ABB RAPID module: WeldProgram.mod

MODULE WeldProgram

    ! =========================
    ! ======= SAFE POS ========
    ! =========================
    PERS robtarget pSafeS1 := [[82.84,919.33,1175.90],[0.326608,0.635474,-0.637382,0.288521],[0,0,-1,0],[9E9,9E9,9E9,9E9,9E9,9E9]];
    PERS robtarget pSafeS1Weld := [[82.84,919.33,1175.90],[0.326608,0.635474,-0.637382,0.288521],[0,0,-1,0],[9E9,9E9,9E9,9E9,9E9,9E9]];
    PERS robtarget pSetup  := [[82.84,919.33,1175.90],[0.326608,0.635474,-0.637382,0.288521],[0,0,-1,0],[9E9,9E9,9E9,9E9,9E9,9E9]];
    PERS robtarget pBullseye := [[82.84,919.33,1175.90],[0.326608,0.635474,-0.637382,0.288521],[0,0,-1,0],[9E9,9E9,9E9,9E9,9E9,9E9]];
    PERS robtarget pFixtureCheck := [[82.84,919.33,1175.90],[0.326608,0.635474,-0.637382,0.288521],[0,0,-1,0],[9E9,9E9,9E9,9E9,9E9,9E9]];

    ! =========================
    ! == DEFAULT WELD DATA ====
    ! =========================
    PERS seamdata cSeamDefault := [1,1,[1,0,14,127,0,0,0,0,0],0,0,0,0,0,[0,0,0,0,0,0,0,0,0],0,0,[0,0,0,0,0,0,0,0,0],0,0,[0,0,0,0,0,0,0,0,0],0];
    PERS welddata cWeldDefault := [6.90033,6.90033,[1,0,19,110.71,0,0,0,0,0],[0,0,18.5,110.71,0,0,0,0,0]];
    PERS weavedata cWeaveDefault := [1,1,3.81,5.08,1.778,0,0,0,0,0,0,0,0,0,0];

    ! =========================
    ! === PART METADATA =======
    ! =========================
    PERS string partNameP01 := "Part 1";
    PERS string partNameP02 := "Part 2";
    PERS string partNameP03 := "Part 3";
    PERS string partNameP04 := "Part 4";
    PERS string partNameP05 := "Part 5";
    PERS string partNameP06 := "Part 6";
    PERS bool partEnabledP01 := TRUE;
    PERS bool partEnabledP02 := TRUE;
    PERS bool partEnabledP03 := TRUE;
    PERS bool partEnabledP04 := TRUE;
    PERS bool partEnabledP05 := TRUE;
    PERS bool partEnabledP06 := TRUE;

    ! =========================
    ! ====== SPEEDS ===========
    ! =========================
    PERS speeddata vPreviewArcStart := [5,500,5000,1000];
    PERS speeddata vPreviewArcEnd := [5,500,5000,1000];
    PERS speeddata vPreviewApproach := [5,500,5000,1000];
    PERS speeddata vPreviewRetract := [5,500,5000,1000];
    PERS speeddata vPreviewTrans := [5,500,5000,1000];
    PERS speeddata vProdArcStart := [100,500,5000,1000];
    PERS speeddata vProdArcEnd := [100,500,5000,1000];
    PERS speeddata vProdApproach := [100,500,5000,1000];
    PERS speeddata vProdRetract := [100,500,5000,1000];
    PERS speeddata vProdTrans := [100,500,5000,1000];

    ! =========================
    ! == ORIENTATION POSES ====
    ! =========================
    PERS robtarget pOri_Left := [[-322.341,524.952,62.8015],[0.119487,0.856675,-0.263973,0.426789],[1,-1,-1,0],[9E+09,9E+09,9E+09,9E+09,9E+09,9E+09]];
    PERS robtarget pOri_Right:= [[-338.053,523.699,62.2846],[0.437822,0.2846,-0.843699,0.124444],[1,0,0,0],[9E+09,9E+09,9E+09,9E+09,9E+09,9E+09]];
    PERS robtarget pOri_Up   := [[-324.994,521.603,62.1105],[0.180394,0.831672,-0.360019,0.382317],[1,0,-1,0],[9E+09,9E+09,9E+09,9E+09,9E+09,9E+09]];
    PERS robtarget pOri_Down := [[-327.638,525.763,56.7062],[0.26234,-0.322639,0.903337,0.105184],[1,-1,2,0],[9E+09,9E+09,9E+09,9E+09,9E+09,9E+09]];
    PERS robtarget pOri_yMid := [[0,0,0],[1,0,0,0],[0,0,0,0],[9E9,9E9,9E9,9E9,9E9,9E9]];
    PERS robtarget pOri_xMid := [[0,0,0],[1,0,0,0],[0,0,0,0],[9E9,9E9,9E9,9E9,9E9,9E9]];

    ! =========================
    ! ===== PART FRAMES =======
    ! =========================
    PERS robtarget P01Origin := [[0,0,0],[1,0,0,0],[0,0,0,0],[9E9,9E9,9E9,9E9,9E9,9E9]];
    PERS robtarget P01Max    := [[0,0,0],[1,0,0,0],[0,0,0,0],[9E9,9E9,9E9,9E9,9E9,9E9]];
    PERS robtarget P01Zoff   := [[0,0,0],[1,0,0,0],[0,0,0,0],[9E9,9E9,9E9,9E9,9E9,9E9]];
    PERS wobjdata wobjP01 := [FALSE,TRUE,"",[[0,0,0],[1,0,0,0]],[[0,0,0],[1,0,0,0]]];
    PERS num nWeldsP01 := 5;

    PERS robtarget P02Origin := [[-1364.6,652.519,70.0999],[0.0320518,0.697908,-0.715468,-0.00179197],[1,-1,1,0],[9E+09,9E+09,9E+09,9E+09,9E+09,9E+09]];
    PERS robtarget P02Max    := [[-382.936,1483.05,51.6185],[0.0320653,0.697883,-0.715492,-0.00180713],[1,-2,1,0],[9E+09,9E+09,9E+09,9E+09,9E+09,9E+09]];
    PERS robtarget P02Zoff   := [[-392.282,1373.57,51.6146],[0.032034,0.697931,-0.715446,-0.00178465],[1,-2,1,0],[9E+09,9E+09,9E+09,9E+09,9E+09,9E+09]];
    PERS wobjdata wobjP02 := [FALSE,TRUE,"",[[-1364.6,652.519,70.0999],[0.0320518,0.697908,-0.715468,-0.00179197]],[[-392.282,1373.57,51.6146],[0.032034,0.697931,-0.715446,-0.00178465]]];
    PERS num nWeldsP02 := 2;

    PERS robtarget P03Origin := [[0,0,0],[1,0,0,0],[0,0,0,0],[9E9,9E9,9E9,9E9,9E9,9E9]];
    PERS robtarget P03Max    := [[0,0,0],[1,0,0,0],[0,0,0,0],[9E9,9E9,9E9,9E9,9E9,9E9]];
    PERS robtarget P03Zoff   := [[0,0,0],[1,0,0,0],[0,0,0,0],[9E9,9E9,9E9,9E9,9E9,9E9]];
    PERS wobjdata wobjP03 := [FALSE,TRUE,"",[[0,0,0],[1,0,0,0]],[[0,0,0],[1,0,0,0]]];
    PERS num nWeldsP03 := 0;

    PERS robtarget P04Origin := [[0,0,0],[1,0,0,0],[0,0,0,0],[9E9,9E9,9E9,9E9,9E9,9E9]];
    PERS robtarget P04Max    := [[0,0,0],[1,0,0,0],[0,0,0,0],[9E9,9E9,9E9,9E9,9E9,9E9]];
    PERS robtarget P04Zoff   := [[0,0,0],[1,0,0,0],[0,0,0,0],[9E9,9E9,9E9,9E9,9E9,9E9]];
    PERS wobjdata wobjP04 := [FALSE,TRUE,"",[[0,0,0],[1,0,0,0]],[[0,0,0],[1,0,0,0]]];
    PERS num nWeldsP04 := 0;

    PERS robtarget P05Origin := [[0,0,0],[1,0,0,0],[0,0,0,0],[9E9,9E9,9E9,9E9,9E9,9E9]];
    PERS robtarget P05Max    := [[0,0,0],[1,0,0,0],[0,0,0,0],[9E9,9E9,9E9,9E9,9E9,9E9]];
    PERS robtarget P05Zoff   := [[0,0,0],[1,0,0,0],[0,0,0,0],[9E9,9E9,9E9,9E9,9E9,9E9]];
    PERS wobjdata wobjP05 := [FALSE,TRUE,"",[[0,0,0],[1,0,0,0]],[[0,0,0],[1,0,0,0]]];
    PERS num nWeldsP05 := 0;

    PERS robtarget P06Origin := [[0,0,0],[1,0,0,0],[0,0,0,0],[9E9,9E9,9E9,9E9,9E9,9E9]];
    PERS robtarget P06Max    := [[0,0,0],[1,0,0,0],[0,0,0,0],[9E9,9E9,9E9,9E9,9E9,9E9]];
    PERS robtarget P06Zoff   := [[0,0,0],[1,0,0,0],[0,0,0,0],[9E9,9E9,9E9,9E9,9E9,9E9]];
    PERS wobjdata wobjP06 := [FALSE,TRUE,"",[[0,0,0],[1,0,0,0]],[[0,0,0],[1,0,0,0]]];
    PERS num nWeldsP06 := 0;

    ! =========================
    ! == WELD SLOT STORAGE ====
    ! =========================
    ! ---- P01 weld slots ----
    PERS bool P01W01_Used := TRUE;
    PERS num  P01W01_SubType := 22;
    PERS num  P01W01_ToolSel := 4;
    PERS num  P01W01_LenMM := 31.75;
    PERS robtarget P01W01_ArcStart := [[-1.72108,1549.32,-10.8357],[0.26234,-0.322639,0.903337,0.105184],[1,-1,2,0],[9E+09,9E+09,9E+09,9E+09,9E+09,9E+09]];
    PERS robtarget P01W01_ArcEnd   := [[30.0289,1549.32,-10.8357],[0.26234,-0.322639,0.903337,0.105184],[1,-1,2,0],[9E+09,9E+09,9E+09,9E+09,9E+09,9E+09]];
    PERS robtarget P01W01_Approach := [[-4.26108,1546.78,-8.29572],[0.26234,-0.322639,0.903337,0.105184],[1,-1,2,0],[9E+09,9E+09,9E+09,9E+09,9E+09,9E+09]];
    PERS robtarget P01W01_Retract  := [[27.4889,1546.78,-8.29572],[0.26234,-0.322639,0.903337,0.105184],[1,-1,2,0],[9E+09,9E+09,9E+09,9E+09,9E+09,9E+09]];
    PERS robtarget P01W01_Trans    := [[27.4889,1546.78,245.704],[0.26234,-0.322639,0.903337,0.105184],[1,-1,2,0],[9E+09,9E+09,9E+09,9E+09,9E+09,9E+09]];
    PERS bool P01W02_Used := TRUE;
    PERS num  P01W02_SubType := 21;
    PERS num  P01W02_ToolSel := 3;
    PERS num  P01W02_LenMM := 31.75;
    PERS robtarget P01W02_ArcStart := [[-313.218,545.116,2.61322],[0.180394,0.831672,-0.360019,0.382317],[1,0,-1,0],[9E+09,9E+09,9E+09,9E+09,9E+09,9E+09]];
    PERS robtarget P01W02_ArcEnd   := [[-281.468,545.116,2.61322],[0.180394,0.831672,-0.360019,0.382317],[1,0,-1,0],[9E+09,9E+09,9E+09,9E+09,9E+09,9E+09]];
    PERS robtarget P01W02_Approach := [[-315.758,547.656,5.15322],[0.180394,0.831672,-0.360019,0.382317],[1,0,-1,0],[9E+09,9E+09,9E+09,9E+09,9E+09,9E+09]];
    PERS robtarget P01W02_Retract  := [[-284.008,547.656,5.15322],[0.180394,0.831672,-0.360019,0.382317],[1,0,-1,0],[9E+09,9E+09,9E+09,9E+09,9E+09,9E+09]];
    PERS robtarget P01W02_Trans    := [[-284.008,547.656,259.153],[0.180394,0.831672,-0.360019,0.382317],[1,0,-1,0],[9E+09,9E+09,9E+09,9E+09,9E+09,9E+09]];
    PERS bool P01W03_Used := TRUE;
    PERS num  P01W03_SubType := 21;
    PERS num  P01W03_ToolSel := 3;
    PERS num  P01W03_LenMM := 31.75;
    PERS robtarget P01W03_ArcStart := [[4.28168,545.116,2.61322],[0.180394,0.831672,-0.360019,0.382317],[1,0,-1,0],[9E+09,9E+09,9E+09,9E+09,9E+09,9E+09]];
    PERS robtarget P01W03_ArcEnd   := [[36.0317,545.116,2.61322],[0.180394,0.831672,-0.360019,0.382317],[1,0,-1,0],[9E+09,9E+09,9E+09,9E+09,9E+09,9E+09]];
    PERS robtarget P01W03_Approach := [[1.74168,547.656,5.15322],[0.180394,0.831672,-0.360019,0.382317],[1,0,-1,0],[9E+09,9E+09,9E+09,9E+09,9E+09,9E+09]];
    PERS robtarget P01W03_Retract  := [[33.4917,547.656,5.15322],[0.180394,0.831672,-0.360019,0.382317],[1,0,-1,0],[9E+09,9E+09,9E+09,9E+09,9E+09,9E+09]];
    PERS robtarget P01W03_Trans    := [[33.4917,547.656,259.153],[0.180394,0.831672,-0.360019,0.382317],[1,0,-1,0],[9E+09,9E+09,9E+09,9E+09,9E+09,9E+09]];
    PERS bool P01W04_Used := TRUE;
    PERS num  P01W04_SubType := 21;
    PERS num  P01W04_ToolSel := 3;
    PERS num  P01W04_LenMM := 31.75;
    PERS robtarget P01W04_ArcStart := [[861.532,545.116,2.61322],[0.180394,0.831672,-0.360019,0.382317],[1,0,-1,0],[9E+09,9E+09,9E+09,9E+09,9E+09,9E+09]];
    PERS robtarget P01W04_ArcEnd   := [[893.282,545.116,2.61322],[0.180394,0.831672,-0.360019,0.382317],[1,0,-1,0],[9E+09,9E+09,9E+09,9E+09,9E+09,9E+09]];
    PERS robtarget P01W04_Approach := [[858.992,547.656,5.15322],[0.180394,0.831672,-0.360019,0.382317],[1,0,-1,0],[9E+09,9E+09,9E+09,9E+09,9E+09,9E+09]];
    PERS robtarget P01W04_Retract  := [[890.742,547.656,5.15322],[0.180394,0.831672,-0.360019,0.382317],[1,0,-1,0],[9E+09,9E+09,9E+09,9E+09,9E+09,9E+09]];
    PERS robtarget P01W04_Trans    := [[890.742,547.656,259.153],[0.180394,0.831672,-0.360019,0.382317],[1,0,-1,0],[9E+09,9E+09,9E+09,9E+09,9E+09,9E+09]];
    PERS bool P01W05_Used := TRUE;
    PERS num  P01W05_SubType := 21;
    PERS num  P01W05_ToolSel := 3;
    PERS num  P01W05_LenMM := 31.75;
    PERS robtarget P01W05_ArcStart := [[1166.33,545.116,2.61322],[0.180394,0.831672,-0.360019,0.382317],[1,0,-1,0],[9E+09,9E+09,9E+09,9E+09,9E+09,9E+09]];
    PERS robtarget P01W05_ArcEnd   := [[1198.08,545.116,2.61322],[0.180394,0.831672,-0.360019,0.382317],[1,0,-1,0],[9E+09,9E+09,9E+09,9E+09,9E+09,9E+09]];
    PERS robtarget P01W05_Approach := [[1163.79,547.656,5.15322],[0.180394,0.831672,-0.360019,0.382317],[1,0,-1,0],[9E+09,9E+09,9E+09,9E+09,9E+09,9E+09]];
    PERS robtarget P01W05_Retract  := [[1195.54,547.656,5.15322],[0.180394,0.831672,-0.360019,0.382317],[1,0,-1,0],[9E+09,9E+09,9E+09,9E+09,9E+09,9E+09]];
    PERS robtarget P01W05_Trans    := [[1195.54,547.656,259.153],[0.180394,0.831672,-0.360019,0.382317],[1,0,-1,0],[9E+09,9E+09,9E+09,9E+09,9E+09,9E+09]];
    PERS bool P01W06_Used := FALSE;
    PERS num  P01W06_SubType := 0;
    PERS num  P01W06_ToolSel := 0;
    PERS num  P01W06_LenMM := 0;
    PERS robtarget P01W06_ArcStart := [[0,0,0],[1,0,0,0],[0,0,0,0],[9E9,9E9,9E9,9E9,9E9,9E9]];
    PERS robtarget P01W06_ArcEnd   := [[0,0,0],[1,0,0,0],[0,0,0,0],[9E9,9E9,9E9,9E9,9E9,9E9]];
    PERS robtarget P01W06_Approach := [[0,0,0],[1,0,0,0],[0,0,0,0],[9E9,9E9,9E9,9E9,9E9,9E9]];
    PERS robtarget P01W06_Retract  := [[0,0,0],[1,0,0,0],[0,0,0,0],[9E9,9E9,9E9,9E9,9E9,9E9]];
    PERS robtarget P01W06_Trans    := [[0,0,0],[1,0,0,0],[0,0,0,0],[9E9,9E9,9E9,9E9,9E9,9E9]];
    PERS bool P01W07_Used := FALSE;
    PERS num  P01W07_SubType := 0;
    PERS num  P01W07_ToolSel := 0;
    PERS num  P01W07_LenMM := 0;
    PERS robtarget P01W07_ArcStart := [[0,0,0],[1,0,0,0],[0,0,0,0],[9E9,9E9,9E9,9E9,9E9,9E9]];
    PERS robtarget P01W07_ArcEnd   := [[0,0,0],[1,0,0,0],[0,0,0,0],[9E9,9E9,9E9,9E9,9E9,9E9]];
    PERS robtarget P01W07_Approach := [[0,0,0],[1,0,0,0],[0,0,0,0],[9E9,9E9,9E9,9E9,9E9,9E9]];
    PERS robtarget P01W07_Retract  := [[0,0,0],[1,0,0,0],[0,0,0,0],[9E9,9E9,9E9,9E9,9E9,9E9]];
    PERS robtarget P01W07_Trans    := [[0,0,0],[1,0,0,0],[0,0,0,0],[9E9,9E9,9E9,9E9,9E9,9E9]];
    PERS bool P01W08_Used := FALSE;
    PERS num  P01W08_SubType := 0;
    PERS num  P01W08_ToolSel := 0;
    PERS num  P01W08_LenMM := 0;
    PERS robtarget P01W08_ArcStart := [[0,0,0],[1,0,0,0],[0,0,0,0],[9E9,9E9,9E9,9E9,9E9,9E9]];
    PERS robtarget P01W08_ArcEnd   := [[0,0,0],[1,0,0,0],[0,0,0,0],[9E9,9E9,9E9,9E9,9E9,9E9]];
    PERS robtarget P01W08_Approach := [[0,0,0],[1,0,0,0],[0,0,0,0],[9E9,9E9,9E9,9E9,9E9,9E9]];
    PERS robtarget P01W08_Retract  := [[0,0,0],[1,0,0,0],[0,0,0,0],[9E9,9E9,9E9,9E9,9E9,9E9]];
    PERS robtarget P01W08_Trans    := [[0,0,0],[1,0,0,0],[0,0,0,0],[9E9,9E9,9E9,9E9,9E9,9E9]];
    PERS bool P01W09_Used := FALSE;
    PERS num  P01W09_SubType := 0;
    PERS num  P01W09_ToolSel := 0;
    PERS num  P01W09_LenMM := 0;
    PERS robtarget P01W09_ArcStart := [[0,0,0],[1,0,0,0],[0,0,0,0],[9E9,9E9,9E9,9E9,9E9,9E9]];
    PERS robtarget P01W09_ArcEnd   := [[0,0,0],[1,0,0,0],[0,0,0,0],[9E9,9E9,9E9,9E9,9E9,9E9]];
    PERS robtarget P01W09_Approach := [[0,0,0],[1,0,0,0],[0,0,0,0],[9E9,9E9,9E9,9E9,9E9,9E9]];
    PERS robtarget P01W09_Retract  := [[0,0,0],[1,0,0,0],[0,0,0,0],[9E9,9E9,9E9,9E9,9E9,9E9]];
    PERS robtarget P01W09_Trans    := [[0,0,0],[1,0,0,0],[0,0,0,0],[9E9,9E9,9E9,9E9,9E9,9E9]];
    PERS bool P01W10_Used := FALSE;
    PERS num  P01W10_SubType := 0;
    PERS num  P01W10_ToolSel := 0;
    PERS num  P01W10_LenMM := 0;
    PERS robtarget P01W10_ArcStart := [[0,0,0],[1,0,0,0],[0,0,0,0],[9E9,9E9,9E9,9E9,9E9,9E9]];
    PERS robtarget P01W10_ArcEnd   := [[0,0,0],[1,0,0,0],[0,0,0,0],[9E9,9E9,9E9,9E9,9E9,9E9]];
    PERS robtarget P01W10_Approach := [[0,0,0],[1,0,0,0],[0,0,0,0],[9E9,9E9,9E9,9E9,9E9,9E9]];
    PERS robtarget P01W10_Retract  := [[0,0,0],[1,0,0,0],[0,0,0,0],[9E9,9E9,9E9,9E9,9E9,9E9]];
    PERS robtarget P01W10_Trans    := [[0,0,0],[1,0,0,0],[0,0,0,0],[9E9,9E9,9E9,9E9,9E9,9E9]];
    PERS bool P01W11_Used := FALSE;
    PERS num  P01W11_SubType := 0;
    PERS num  P01W11_ToolSel := 0;
    PERS num  P01W11_LenMM := 0;
    PERS robtarget P01W11_ArcStart := [[0,0,0],[1,0,0,0],[0,0,0,0],[9E9,9E9,9E9,9E9,9E9,9E9]];
    PERS robtarget P01W11_ArcEnd   := [[0,0,0],[1,0,0,0],[0,0,0,0],[9E9,9E9,9E9,9E9,9E9,9E9]];
    PERS robtarget P01W11_Approach := [[0,0,0],[1,0,0,0],[0,0,0,0],[9E9,9E9,9E9,9E9,9E9,9E9]];
    PERS robtarget P01W11_Retract  := [[0,0,0],[1,0,0,0],[0,0,0,0],[9E9,9E9,9E9,9E9,9E9,9E9]];
    PERS robtarget P01W11_Trans    := [[0,0,0],[1,0,0,0],[0,0,0,0],[9E9,9E9,9E9,9E9,9E9,9E9]];
    PERS bool P01W12_Used := FALSE;
    PERS num  P01W12_SubType := 0;
    PERS num  P01W12_ToolSel := 0;
    PERS num  P01W12_LenMM := 0;
    PERS robtarget P01W12_ArcStart := [[0,0,0],[1,0,0,0],[0,0,0,0],[9E9,9E9,9E9,9E9,9E9,9E9]];
    PERS robtarget P01W12_ArcEnd   := [[0,0,0],[1,0,0,0],[0,0,0,0],[9E9,9E9,9E9,9E9,9E9,9E9]];
    PERS robtarget P01W12_Approach := [[0,0,0],[1,0,0,0],[0,0,0,0],[9E9,9E9,9E9,9E9,9E9,9E9]];
    PERS robtarget P01W12_Retract  := [[0,0,0],[1,0,0,0],[0,0,0,0],[9E9,9E9,9E9,9E9,9E9,9E9]];
    PERS robtarget P01W12_Trans    := [[0,0,0],[1,0,0,0],[0,0,0,0],[9E9,9E9,9E9,9E9,9E9,9E9]];
    PERS bool P01W13_Used := FALSE;
    PERS num  P01W13_SubType := 0;
    PERS num  P01W13_ToolSel := 0;
    PERS num  P01W13_LenMM := 0;
    PERS robtarget P01W13_ArcStart := [[0,0,0],[1,0,0,0],[0,0,0,0],[9E9,9E9,9E9,9E9,9E9,9E9]];
    PERS robtarget P01W13_ArcEnd   := [[0,0,0],[1,0,0,0],[0,0,0,0],[9E9,9E9,9E9,9E9,9E9,9E9]];
    PERS robtarget P01W13_Approach := [[0,0,0],[1,0,0,0],[0,0,0,0],[9E9,9E9,9E9,9E9,9E9,9E9]];
    PERS robtarget P01W13_Retract  := [[0,0,0],[1,0,0,0],[0,0,0,0],[9E9,9E9,9E9,9E9,9E9,9E9]];
    PERS robtarget P01W13_Trans    := [[0,0,0],[1,0,0,0],[0,0,0,0],[9E9,9E9,9E9,9E9,9E9,9E9]];
    PERS bool P01W14_Used := FALSE;
    PERS num  P01W14_SubType := 0;
    PERS num  P01W14_ToolSel := 0;
    PERS num  P01W14_LenMM := 0;
    PERS robtarget P01W14_ArcStart := [[0,0,0],[1,0,0,0],[0,0,0,0],[9E9,9E9,9E9,9E9,9E9,9E9]];
    PERS robtarget P01W14_ArcEnd   := [[0,0,0],[1,0,0,0],[0,0,0,0],[9E9,9E9,9E9,9E9,9E9,9E9]];
    PERS robtarget P01W14_Approach := [[0,0,0],[1,0,0,0],[0,0,0,0],[9E9,9E9,9E9,9E9,9E9,9E9]];
    PERS robtarget P01W14_Retract  := [[0,0,0],[1,0,0,0],[0,0,0,0],[9E9,9E9,9E9,9E9,9E9,9E9]];
    PERS robtarget P01W14_Trans    := [[0,0,0],[1,0,0,0],[0,0,0,0],[9E9,9E9,9E9,9E9,9E9,9E9]];
    PERS bool P01W15_Used := FALSE;
    PERS num  P01W15_SubType := 0;
    PERS num  P01W15_ToolSel := 0;
    PERS num  P01W15_LenMM := 0;
    PERS robtarget P01W15_ArcStart := [[0,0,0],[1,0,0,0],[0,0,0,0],[9E9,9E9,9E9,9E9,9E9,9E9]];
    PERS robtarget P01W15_ArcEnd   := [[0,0,0],[1,0,0,0],[0,0,0,0],[9E9,9E9,9E9,9E9,9E9,9E9]];
    PERS robtarget P01W15_Approach := [[0,0,0],[1,0,0,0],[0,0,0,0],[9E9,9E9,9E9,9E9,9E9,9E9]];
    PERS robtarget P01W15_Retract  := [[0,0,0],[1,0,0,0],[0,0,0,0],[9E9,9E9,9E9,9E9,9E9,9E9]];
    PERS robtarget P01W15_Trans    := [[0,0,0],[1,0,0,0],[0,0,0,0],[9E9,9E9,9E9,9E9,9E9,9E9]];
    PERS bool P01W16_Used := FALSE;
    PERS num  P01W16_SubType := 0;
    PERS num  P01W16_ToolSel := 0;
    PERS num  P01W16_LenMM := 0;
    PERS robtarget P01W16_ArcStart := [[0,0,0],[1,0,0,0],[0,0,0,0],[9E9,9E9,9E9,9E9,9E9,9E9]];
    PERS robtarget P01W16_ArcEnd   := [[0,0,0],[1,0,0,0],[0,0,0,0],[9E9,9E9,9E9,9E9,9E9,9E9]];
    PERS robtarget P01W16_Approach := [[0,0,0],[1,0,0,0],[0,0,0,0],[9E9,9E9,9E9,9E9,9E9,9E9]];
    PERS robtarget P01W16_Retract  := [[0,0,0],[1,0,0,0],[0,0,0,0],[9E9,9E9,9E9,9E9,9E9,9E9]];
    PERS robtarget P01W16_Trans    := [[0,0,0],[1,0,0,0],[0,0,0,0],[9E9,9E9,9E9,9E9,9E9,9E9]];
    PERS bool P01W17_Used := FALSE;
    PERS num  P01W17_SubType := 0;
    PERS num  P01W17_ToolSel := 0;
    PERS num  P01W17_LenMM := 0;
    PERS robtarget P01W17_ArcStart := [[0,0,0],[1,0,0,0],[0,0,0,0],[9E9,9E9,9E9,9E9,9E9,9E9]];
    PERS robtarget P01W17_ArcEnd   := [[0,0,0],[1,0,0,0],[0,0,0,0],[9E9,9E9,9E9,9E9,9E9,9E9]];
    PERS robtarget P01W17_Approach := [[0,0,0],[1,0,0,0],[0,0,0,0],[9E9,9E9,9E9,9E9,9E9,9E9]];
    PERS robtarget P01W17_Retract  := [[0,0,0],[1,0,0,0],[0,0,0,0],[9E9,9E9,9E9,9E9,9E9,9E9]];
    PERS robtarget P01W17_Trans    := [[0,0,0],[1,0,0,0],[0,0,0,0],[9E9,9E9,9E9,9E9,9E9,9E9]];
    PERS bool P01W18_Used := FALSE;
    PERS num  P01W18_SubType := 0;
    PERS num  P01W18_ToolSel := 0;
    PERS num  P01W18_LenMM := 0;
    PERS robtarget P01W18_ArcStart := [[0,0,0],[1,0,0,0],[0,0,0,0],[9E9,9E9,9E9,9E9,9E9,9E9]];
    PERS robtarget P01W18_ArcEnd   := [[0,0,0],[1,0,0,0],[0,0,0,0],[9E9,9E9,9E9,9E9,9E9,9E9]];
    PERS robtarget P01W18_Approach := [[0,0,0],[1,0,0,0],[0,0,0,0],[9E9,9E9,9E9,9E9,9E9,9E9]];
    PERS robtarget P01W18_Retract  := [[0,0,0],[1,0,0,0],[0,0,0,0],[9E9,9E9,9E9,9E9,9E9,9E9]];
    PERS robtarget P01W18_Trans    := [[0,0,0],[1,0,0,0],[0,0,0,0],[9E9,9E9,9E9,9E9,9E9,9E9]];
    PERS bool P01W19_Used := FALSE;
    PERS num  P01W19_SubType := 0;
    PERS num  P01W19_ToolSel := 0;
    PERS num  P01W19_LenMM := 0;
    PERS robtarget P01W19_ArcStart := [[0,0,0],[1,0,0,0],[0,0,0,0],[9E9,9E9,9E9,9E9,9E9,9E9]];
    PERS robtarget P01W19_ArcEnd   := [[0,0,0],[1,0,0,0],[0,0,0,0],[9E9,9E9,9E9,9E9,9E9,9E9]];
    PERS robtarget P01W19_Approach := [[0,0,0],[1,0,0,0],[0,0,0,0],[9E9,9E9,9E9,9E9,9E9,9E9]];
    PERS robtarget P01W19_Retract  := [[0,0,0],[1,0,0,0],[0,0,0,0],[9E9,9E9,9E9,9E9,9E9,9E9]];
    PERS robtarget P01W19_Trans    := [[0,0,0],[1,0,0,0],[0,0,0,0],[9E9,9E9,9E9,9E9,9E9,9E9]];
    PERS bool P01W20_Used := FALSE;
    PERS num  P01W20_SubType := 0;
    PERS num  P01W20_ToolSel := 0;
    PERS num  P01W20_LenMM := 0;
    PERS robtarget P01W20_ArcStart := [[0,0,0],[1,0,0,0],[0,0,0,0],[9E9,9E9,9E9,9E9,9E9,9E9]];
    PERS robtarget P01W20_ArcEnd   := [[0,0,0],[1,0,0,0],[0,0,0,0],[9E9,9E9,9E9,9E9,9E9,9E9]];
    PERS robtarget P01W20_Approach := [[0,0,0],[1,0,0,0],[0,0,0,0],[9E9,9E9,9E9,9E9,9E9,9E9]];
    PERS robtarget P01W20_Retract  := [[0,0,0],[1,0,0,0],[0,0,0,0],[9E9,9E9,9E9,9E9,9E9,9E9]];
    PERS robtarget P01W20_Trans    := [[0,0,0],[1,0,0,0],[0,0,0,0],[9E9,9E9,9E9,9E9,9E9,9E9]];
    PERS bool P01W21_Used := FALSE;
    PERS num  P01W21_SubType := 0;
    PERS num  P01W21_ToolSel := 0;
    PERS num  P01W21_LenMM := 0;
    PERS robtarget P01W21_ArcStart := [[0,0,0],[1,0,0,0],[0,0,0,0],[9E9,9E9,9E9,9E9,9E9,9E9]];
    PERS robtarget P01W21_ArcEnd   := [[0,0,0],[1,0,0,0],[0,0,0,0],[9E9,9E9,9E9,9E9,9E9,9E9]];
    PERS robtarget P01W21_Approach := [[0,0,0],[1,0,0,0],[0,0,0,0],[9E9,9E9,9E9,9E9,9E9,9E9]];
    PERS robtarget P01W21_Retract  := [[0,0,0],[1,0,0,0],[0,0,0,0],[9E9,9E9,9E9,9E9,9E9,9E9]];
    PERS robtarget P01W21_Trans    := [[0,0,0],[1,0,0,0],[0,0,0,0],[9E9,9E9,9E9,9E9,9E9,9E9]];
    PERS bool P01W22_Used := FALSE;
    PERS num  P01W22_SubType := 0;
    PERS num  P01W22_ToolSel := 0;
    PERS num  P01W22_LenMM := 0;
    PERS robtarget P01W22_ArcStart := [[0,0,0],[1,0,0,0],[0,0,0,0],[9E9,9E9,9E9,9E9,9E9,9E9]];
    PERS robtarget P01W22_ArcEnd   := [[0,0,0],[1,0,0,0],[0,0,0,0],[9E9,9E9,9E9,9E9,9E9,9E9]];
    PERS robtarget P01W22_Approach := [[0,0,0],[1,0,0,0],[0,0,0,0],[9E9,9E9,9E9,9E9,9E9,9E9]];
    PERS robtarget P01W22_Retract  := [[0,0,0],[1,0,0,0],[0,0,0,0],[9E9,9E9,9E9,9E9,9E9,9E9]];
    PERS robtarget P01W22_Trans    := [[0,0,0],[1,0,0,0],[0,0,0,0],[9E9,9E9,9E9,9E9,9E9,9E9]];
    PERS bool P01W23_Used := FALSE;
    PERS num  P01W23_SubType := 0;
    PERS num  P01W23_ToolSel := 0;
    PERS num  P01W23_LenMM := 0;
    PERS robtarget P01W23_ArcStart := [[0,0,0],[1,0,0,0],[0,0,0,0],[9E9,9E9,9E9,9E9,9E9,9E9]];
    PERS robtarget P01W23_ArcEnd   := [[0,0,0],[1,0,0,0],[0,0,0,0],[9E9,9E9,9E9,9E9,9E9,9E9]];
    PERS robtarget P01W23_Approach := [[0,0,0],[1,0,0,0],[0,0,0,0],[9E9,9E9,9E9,9E9,9E9,9E9]];
    PERS robtarget P01W23_Retract  := [[0,0,0],[1,0,0,0],[0,0,0,0],[9E9,9E9,9E9,9E9,9E9,9E9]];
    PERS robtarget P01W23_Trans    := [[0,0,0],[1,0,0,0],[0,0,0,0],[9E9,9E9,9E9,9E9,9E9,9E9]];
    PERS bool P01W24_Used := FALSE;
    PERS num  P01W24_SubType := 0;
    PERS num  P01W24_ToolSel := 0;
    PERS num  P01W24_LenMM := 0;
    PERS robtarget P01W24_ArcStart := [[0,0,0],[1,0,0,0],[0,0,0,0],[9E9,9E9,9E9,9E9,9E9,9E9]];
    PERS robtarget P01W24_ArcEnd   := [[0,0,0],[1,0,0,0],[0,0,0,0],[9E9,9E9,9E9,9E9,9E9,9E9]];
    PERS robtarget P01W24_Approach := [[0,0,0],[1,0,0,0],[0,0,0,0],[9E9,9E9,9E9,9E9,9E9,9E9]];
    PERS robtarget P01W24_Retract  := [[0,0,0],[1,0,0,0],[0,0,0,0],[9E9,9E9,9E9,9E9,9E9,9E9]];
    PERS robtarget P01W24_Trans    := [[0,0,0],[1,0,0,0],[0,0,0,0],[9E9,9E9,9E9,9E9,9E9,9E9]];
    PERS bool P01W25_Used := FALSE;
    PERS num  P01W25_SubType := 0;
    PERS num  P01W25_ToolSel := 0;
    PERS num  P01W25_LenMM := 0;
    PERS robtarget P01W25_ArcStart := [[0,0,0],[1,0,0,0],[0,0,0,0],[9E9,9E9,9E9,9E9,9E9,9E9]];
    PERS robtarget P01W25_ArcEnd   := [[0,0,0],[1,0,0,0],[0,0,0,0],[9E9,9E9,9E9,9E9,9E9,9E9]];
    PERS robtarget P01W25_Approach := [[0,0,0],[1,0,0,0],[0,0,0,0],[9E9,9E9,9E9,9E9,9E9,9E9]];
    PERS robtarget P01W25_Retract  := [[0,0,0],[1,0,0,0],[0,0,0,0],[9E9,9E9,9E9,9E9,9E9,9E9]];
    PERS robtarget P01W25_Trans    := [[0,0,0],[1,0,0,0],[0,0,0,0],[9E9,9E9,9E9,9E9,9E9,9E9]];
    PERS bool P01W26_Used := FALSE;
    PERS num  P01W26_SubType := 0;
    PERS num  P01W26_ToolSel := 0;
    PERS num  P01W26_LenMM := 0;
    PERS robtarget P01W26_ArcStart := [[0,0,0],[1,0,0,0],[0,0,0,0],[9E9,9E9,9E9,9E9,9E9,9E9]];
    PERS robtarget P01W26_ArcEnd   := [[0,0,0],[1,0,0,0],[0,0,0,0],[9E9,9E9,9E9,9E9,9E9,9E9]];
    PERS robtarget P01W26_Approach := [[0,0,0],[1,0,0,0],[0,0,0,0],[9E9,9E9,9E9,9E9,9E9,9E9]];
    PERS robtarget P01W26_Retract  := [[0,0,0],[1,0,0,0],[0,0,0,0],[9E9,9E9,9E9,9E9,9E9,9E9]];
    PERS robtarget P01W26_Trans    := [[0,0,0],[1,0,0,0],[0,0,0,0],[9E9,9E9,9E9,9E9,9E9,9E9]];
    PERS bool P01W27_Used := FALSE;
    PERS num  P01W27_SubType := 0;
    PERS num  P01W27_ToolSel := 0;
    PERS num  P01W27_LenMM := 0;
    PERS robtarget P01W27_ArcStart := [[0,0,0],[1,0,0,0],[0,0,0,0],[9E9,9E9,9E9,9E9,9E9,9E9]];
    PERS robtarget P01W27_ArcEnd   := [[0,0,0],[1,0,0,0],[0,0,0,0],[9E9,9E9,9E9,9E9,9E9,9E9]];
    PERS robtarget P01W27_Approach := [[0,0,0],[1,0,0,0],[0,0,0,0],[9E9,9E9,9E9,9E9,9E9,9E9]];
    PERS robtarget P01W27_Retract  := [[0,0,0],[1,0,0,0],[0,0,0,0],[9E9,9E9,9E9,9E9,9E9,9E9]];
    PERS robtarget P01W27_Trans    := [[0,0,0],[1,0,0,0],[0,0,0,0],[9E9,9E9,9E9,9E9,9E9,9E9]];
    PERS bool P01W28_Used := FALSE;
    PERS num  P01W28_SubType := 0;
    PERS num  P01W28_ToolSel := 0;
    PERS num  P01W28_LenMM := 0;
    PERS robtarget P01W28_ArcStart := [[0,0,0],[1,0,0,0],[0,0,0,0],[9E9,9E9,9E9,9E9,9E9,9E9]];
    PERS robtarget P01W28_ArcEnd   := [[0,0,0],[1,0,0,0],[0,0,0,0],[9E9,9E9,9E9,9E9,9E9,9E9]];
    PERS robtarget P01W28_Approach := [[0,0,0],[1,0,0,0],[0,0,0,0],[9E9,9E9,9E9,9E9,9E9,9E9]];
    PERS robtarget P01W28_Retract  := [[0,0,0],[1,0,0,0],[0,0,0,0],[9E9,9E9,9E9,9E9,9E9,9E9]];
    PERS robtarget P01W28_Trans    := [[0,0,0],[1,0,0,0],[0,0,0,0],[9E9,9E9,9E9,9E9,9E9,9E9]];
    PERS bool P01W29_Used := FALSE;
    PERS num  P01W29_SubType := 0;
    PERS num  P01W29_ToolSel := 0;
    PERS num  P01W29_LenMM := 0;
    PERS robtarget P01W29_ArcStart := [[0,0,0],[1,0,0,0],[0,0,0,0],[9E9,9E9,9E9,9E9,9E9,9E9]];
    PERS robtarget P01W29_ArcEnd   := [[0,0,0],[1,0,0,0],[0,0,0,0],[9E9,9E9,9E9,9E9,9E9,9E9]];
    PERS robtarget P01W29_Approach := [[0,0,0],[1,0,0,0],[0,0,0,0],[9E9,9E9,9E9,9E9,9E9,9E9]];
    PERS robtarget P01W29_Retract  := [[0,0,0],[1,0,0,0],[0,0,0,0],[9E9,9E9,9E9,9E9,9E9,9E9]];
    PERS robtarget P01W29_Trans    := [[0,0,0],[1,0,0,0],[0,0,0,0],[9E9,9E9,9E9,9E9,9E9,9E9]];
    PERS bool P01W30_Used := FALSE;
    PERS num  P01W30_SubType := 0;
    PERS num  P01W30_ToolSel := 0;
    PERS num  P01W30_LenMM := 0;
    PERS robtarget P01W30_ArcStart := [[0,0,0],[1,0,0,0],[0,0,0,0],[9E9,9E9,9E9,9E9,9E9,9E9]];
    PERS robtarget P01W30_ArcEnd   := [[0,0,0],[1,0,0,0],[0,0,0,0],[9E9,9E9,9E9,9E9,9E9,9E9]];
    PERS robtarget P01W30_Approach := [[0,0,0],[1,0,0,0],[0,0,0,0],[9E9,9E9,9E9,9E9,9E9,9E9]];
    PERS robtarget P01W30_Retract  := [[0,0,0],[1,0,0,0],[0,0,0,0],[9E9,9E9,9E9,9E9,9E9,9E9]];
    PERS robtarget P01W30_Trans    := [[0,0,0],[1,0,0,0],[0,0,0,0],[9E9,9E9,9E9,9E9,9E9,9E9]];

    ! ---- P02 weld slots ----
    PERS bool P02W01_Used := TRUE;
    PERS num  P02W01_SubType := 11;
    PERS num  P02W01_ToolSel := 1;
    PERS num  P02W01_LenMM := 19.05;
    PERS robtarget P02W01_ArcStart := [[-1288.01,701.443,82.7337],[0.119487,0.856675,-0.263973,0.426789],[1,-1,-1,0],[9E+09,9E+09,9E+09,9E+09,9E+09,9E+09]];
    PERS robtarget P02W01_ArcEnd   := [[-1288.01,682.393,82.7337],[0.119487,0.856675,-0.263973,0.426789],[1,-1,-1,0],[9E+09,9E+09,9E+09,9E+09,9E+09,9E+09]];
    PERS robtarget P02W01_Approach := [[-1290.55,703.983,85.2737],[0.119487,0.856675,-0.263973,0.426789],[1,-1,-1,0],[9E+09,9E+09,9E+09,9E+09,9E+09,9E+09]];
    PERS robtarget P02W01_Retract  := [[-1290.55,684.933,85.2737],[0.119487,0.856675,-0.263973,0.426789],[1,-1,-1,0],[9E+09,9E+09,9E+09,9E+09,9E+09,9E+09]];
    PERS robtarget P02W01_Trans    := [[-1290.55,684.933,339.274],[0.119487,0.856675,-0.263973,0.426789],[1,-1,-1,0],[9E+09,9E+09,9E+09,9E+09,9E+09,9E+09]];
    PERS bool P02W02_Used := TRUE;
    PERS num  P02W02_SubType := 21;
    PERS num  P02W02_ToolSel := 3;
    PERS num  P02W02_LenMM := 19.05;
    PERS robtarget P02W02_ArcStart := [[-1288.01,701.443,82.7337],[0.180394,0.831672,-0.360019,0.382317],[1,0,-1,0],[9E+09,9E+09,9E+09,9E+09,9E+09,9E+09]];
    PERS robtarget P02W02_ArcEnd   := [[-1268.96,701.443,82.7337],[0.180394,0.831672,-0.360019,0.382317],[1,0,-1,0],[9E+09,9E+09,9E+09,9E+09,9E+09,9E+09]];
    PERS robtarget P02W02_Approach := [[-1290.55,703.983,85.2737],[0.180394,0.831672,-0.360019,0.382317],[1,0,-1,0],[9E+09,9E+09,9E+09,9E+09,9E+09,9E+09]];
    PERS robtarget P02W02_Retract  := [[-1271.5,703.983,85.2737],[0.180394,0.831672,-0.360019,0.382317],[1,0,-1,0],[9E+09,9E+09,9E+09,9E+09,9E+09,9E+09]];
    PERS robtarget P02W02_Trans    := [[-1271.5,703.983,339.274],[0.180394,0.831672,-0.360019,0.382317],[1,0,-1,0],[9E+09,9E+09,9E+09,9E+09,9E+09,9E+09]];
    PERS bool P02W03_Used := FALSE;
    PERS num  P02W03_SubType := 0;
    PERS num  P02W03_ToolSel := 0;
    PERS num  P02W03_LenMM := 0;
    PERS robtarget P02W03_ArcStart := [[0,0,0],[1,0,0,0],[0,0,0,0],[9E9,9E9,9E9,9E9,9E9,9E9]];
    PERS robtarget P02W03_ArcEnd   := [[0,0,0],[1,0,0,0],[0,0,0,0],[9E9,9E9,9E9,9E9,9E9,9E9]];
    PERS robtarget P02W03_Approach := [[0,0,0],[1,0,0,0],[0,0,0,0],[9E9,9E9,9E9,9E9,9E9,9E9]];
    PERS robtarget P02W03_Retract  := [[0,0,0],[1,0,0,0],[0,0,0,0],[9E9,9E9,9E9,9E9,9E9,9E9]];
    PERS robtarget P02W03_Trans    := [[0,0,0],[1,0,0,0],[0,0,0,0],[9E9,9E9,9E9,9E9,9E9,9E9]];
    PERS bool P02W04_Used := FALSE;
    PERS num  P02W04_SubType := 0;
    PERS num  P02W04_ToolSel := 0;
    PERS num  P02W04_LenMM := 0;
    PERS robtarget P02W04_ArcStart := [[0,0,0],[1,0,0,0],[0,0,0,0],[9E9,9E9,9E9,9E9,9E9,9E9]];
    PERS robtarget P02W04_ArcEnd   := [[0,0,0],[1,0,0,0],[0,0,0,0],[9E9,9E9,9E9,9E9,9E9,9E9]];
    PERS robtarget P02W04_Approach := [[0,0,0],[1,0,0,0],[0,0,0,0],[9E9,9E9,9E9,9E9,9E9,9E9]];
    PERS robtarget P02W04_Retract  := [[0,0,0],[1,0,0,0],[0,0,0,0],[9E9,9E9,9E9,9E9,9E9,9E9]];
    PERS robtarget P02W04_Trans    := [[0,0,0],[1,0,0,0],[0,0,0,0],[9E9,9E9,9E9,9E9,9E9,9E9]];
    PERS bool P02W05_Used := FALSE;
    PERS num  P02W05_SubType := 0;
    PERS num  P02W05_ToolSel := 0;
    PERS num  P02W05_LenMM := 0;
    PERS robtarget P02W05_ArcStart := [[0,0,0],[1,0,0,0],[0,0,0,0],[9E9,9E9,9E9,9E9,9E9,9E9]];
    PERS robtarget P02W05_ArcEnd   := [[0,0,0],[1,0,0,0],[0,0,0,0],[9E9,9E9,9E9,9E9,9E9,9E9]];
    PERS robtarget P02W05_Approach := [[0,0,0],[1,0,0,0],[0,0,0,0],[9E9,9E9,9E9,9E9,9E9,9E9]];
    PERS robtarget P02W05_Retract  := [[0,0,0],[1,0,0,0],[0,0,0,0],[9E9,9E9,9E9,9E9,9E9,9E9]];
    PERS robtarget P02W05_Trans    := [[0,0,0],[1,0,0,0],[0,0,0,0],[9E9,9E9,9E9,9E9,9E9,9E9]];
    PERS bool P02W06_Used := FALSE;
    PERS num  P02W06_SubType := 0;
    PERS num  P02W06_ToolSel := 0;
    PERS num  P02W06_LenMM := 0;
    PERS robtarget P02W06_ArcStart := [[0,0,0],[1,0,0,0],[0,0,0,0],[9E9,9E9,9E9,9E9,9E9,9E9]];
    PERS robtarget P02W06_ArcEnd   := [[0,0,0],[1,0,0,0],[0,0,0,0],[9E9,9E9,9E9,9E9,9E9,9E9]];
    PERS robtarget P02W06_Approach := [[0,0,0],[1,0,0,0],[0,0,0,0],[9E9,9E9,9E9,9E9,9E9,9E9]];
    PERS robtarget P02W06_Retract  := [[0,0,0],[1,0,0,0],[0,0,0,0],[9E9,9E9,9E9,9E9,9E9,9E9]];
    PERS robtarget P02W06_Trans    := [[0,0,0],[1,0,0,0],[0,0,0,0],[9E9,9E9,9E9,9E9,9E9,9E9]];
    PERS bool P02W07_Used := FALSE;
    PERS num  P02W07_SubType := 0;
    PERS num  P02W07_ToolSel := 0;
    PERS num  P02W07_LenMM := 0;
    PERS robtarget P02W07_ArcStart := [[0,0,0],[1,0,0,0],[0,0,0,0],[9E9,9E9,9E9,9E9,9E9,9E9]];
    PERS robtarget P02W07_ArcEnd   := [[0,0,0],[1,0,0,0],[0,0,0,0],[9E9,9E9,9E9,9E9,9E9,9E9]];
    PERS robtarget P02W07_Approach := [[0,0,0],[1,0,0,0],[0,0,0,0],[9E9,9E9,9E9,9E9,9E9,9E9]];
    PERS robtarget P02W07_Retract  := [[0,0,0],[1,0,0,0],[0,0,0,0],[9E9,9E9,9E9,9E9,9E9,9E9]];
    PERS robtarget P02W07_Trans    := [[0,0,0],[1,0,0,0],[0,0,0,0],[9E9,9E9,9E9,9E9,9E9,9E9]];
    PERS bool P02W08_Used := FALSE;
    PERS num  P02W08_SubType := 0;
    PERS num  P02W08_ToolSel := 0;
    PERS num  P02W08_LenMM := 0;
    PERS robtarget P02W08_ArcStart := [[0,0,0],[1,0,0,0],[0,0,0,0],[9E9,9E9,9E9,9E9,9E9,9E9]];
    PERS robtarget P02W08_ArcEnd   := [[0,0,0],[1,0,0,0],[0,0,0,0],[9E9,9E9,9E9,9E9,9E9,9E9]];
    PERS robtarget P02W08_Approach := [[0,0,0],[1,0,0,0],[0,0,0,0],[9E9,9E9,9E9,9E9,9E9,9E9]];
    PERS robtarget P02W08_Retract  := [[0,0,0],[1,0,0,0],[0,0,0,0],[9E9,9E9,9E9,9E9,9E9,9E9]];
    PERS robtarget P02W08_Trans    := [[0,0,0],[1,0,0,0],[0,0,0,0],[9E9,9E9,9E9,9E9,9E9,9E9]];
    PERS bool P02W09_Used := FALSE;
    PERS num  P02W09_SubType := 0;
    PERS num  P02W09_ToolSel := 0;
    PERS num  P02W09_LenMM := 0;
    PERS robtarget P02W09_ArcStart := [[0,0,0],[1,0,0,0],[0,0,0,0],[9E9,9E9,9E9,9E9,9E9,9E9]];
    PERS robtarget P02W09_ArcEnd   := [[0,0,0],[1,0,0,0],[0,0,0,0],[9E9,9E9,9E9,9E9,9E9,9E9]];
    PERS robtarget P02W09_Approach := [[0,0,0],[1,0,0,0],[0,0,0,0],[9E9,9E9,9E9,9E9,9E9,9E9]];
    PERS robtarget P02W09_Retract  := [[0,0,0],[1,0,0,0],[0,0,0,0],[9E9,9E9,9E9,9E9,9E9,9E9]];
    PERS robtarget P02W09_Trans    := [[0,0,0],[1,0,0,0],[0,0,0,0],[9E9,9E9,9E9,9E9,9E9,9E9]];
    PERS bool P02W10_Used := FALSE;
    PERS num  P02W10_SubType := 0;
    PERS num  P02W10_ToolSel := 0;
    PERS num  P02W10_LenMM := 0;
    PERS robtarget P02W10_ArcStart := [[0,0,0],[1,0,0,0],[0,0,0,0],[9E9,9E9,9E9,9E9,9E9,9E9]];
    PERS robtarget P02W10_ArcEnd   := [[0,0,0],[1,0,0,0],[0,0,0,0],[9E9,9E9,9E9,9E9,9E9,9E9]];
    PERS robtarget P02W10_Approach := [[0,0,0],[1,0,0,0],[0,0,0,0],[9E9,9E9,9E9,9E9,9E9,9E9]];
    PERS robtarget P02W10_Retract  := [[0,0,0],[1,0,0,0],[0,0,0,0],[9E9,9E9,9E9,9E9,9E9,9E9]];
    PERS robtarget P02W10_Trans    := [[0,0,0],[1,0,0,0],[0,0,0,0],[9E9,9E9,9E9,9E9,9E9,9E9]];
    PERS bool P02W11_Used := FALSE;
    PERS num  P02W11_SubType := 0;
    PERS num  P02W11_ToolSel := 0;
    PERS num  P02W11_LenMM := 0;
    PERS robtarget P02W11_ArcStart := [[0,0,0],[1,0,0,0],[0,0,0,0],[9E9,9E9,9E9,9E9,9E9,9E9]];
    PERS robtarget P02W11_ArcEnd   := [[0,0,0],[1,0,0,0],[0,0,0,0],[9E9,9E9,9E9,9E9,9E9,9E9]];
    PERS robtarget P02W11_Approach := [[0,0,0],[1,0,0,0],[0,0,0,0],[9E9,9E9,9E9,9E9,9E9,9E9]];
    PERS robtarget P02W11_Retract  := [[0,0,0],[1,0,0,0],[0,0,0,0],[9E9,9E9,9E9,9E9,9E9,9E9]];
    PERS robtarget P02W11_Trans    := [[0,0,0],[1,0,0,0],[0,0,0,0],[9E9,9E9,9E9,9E9,9E9,9E9]];
    PERS bool P02W12_Used := FALSE;
    PERS num  P02W12_SubType := 0;
    PERS num  P02W12_ToolSel := 0;
    PERS num  P02W12_LenMM := 0;
    PERS robtarget P02W12_ArcStart := [[0,0,0],[1,0,0,0],[0,0,0,0],[9E9,9E9,9E9,9E9,9E9,9E9]];
    PERS robtarget P02W12_ArcEnd   := [[0,0,0],[1,0,0,0],[0,0,0,0],[9E9,9E9,9E9,9E9,9E9,9E9]];
    PERS robtarget P02W12_Approach := [[0,0,0],[1,0,0,0],[0,0,0,0],[9E9,9E9,9E9,9E9,9E9,9E9]];
    PERS robtarget P02W12_Retract  := [[0,0,0],[1,0,0,0],[0,0,0,0],[9E9,9E9,9E9,9E9,9E9,9E9]];
    PERS robtarget P02W12_Trans    := [[0,0,0],[1,0,0,0],[0,0,0,0],[9E9,9E9,9E9,9E9,9E9,9E9]];
    PERS bool P02W13_Used := FALSE;
    PERS num  P02W13_SubType := 0;
    PERS num  P02W13_ToolSel := 0;
    PERS num  P02W13_LenMM := 0;
    PERS robtarget P02W13_ArcStart := [[0,0,0],[1,0,0,0],[0,0,0,0],[9E9,9E9,9E9,9E9,9E9,9E9]];
    PERS robtarget P02W13_ArcEnd   := [[0,0,0],[1,0,0,0],[0,0,0,0],[9E9,9E9,9E9,9E9,9E9,9E9]];
    PERS robtarget P02W13_Approach := [[0,0,0],[1,0,0,0],[0,0,0,0],[9E9,9E9,9E9,9E9,9E9,9E9]];
    PERS robtarget P02W13_Retract  := [[0,0,0],[1,0,0,0],[0,0,0,0],[9E9,9E9,9E9,9E9,9E9,9E9]];
    PERS robtarget P02W13_Trans    := [[0,0,0],[1,0,0,0],[0,0,0,0],[9E9,9E9,9E9,9E9,9E9,9E9]];
    PERS bool P02W14_Used := FALSE;
    PERS num  P02W14_SubType := 0;
    PERS num  P02W14_ToolSel := 0;
    PERS num  P02W14_LenMM := 0;
    PERS robtarget P02W14_ArcStart := [[0,0,0],[1,0,0,0],[0,0,0,0],[9E9,9E9,9E9,9E9,9E9,9E9]];
    PERS robtarget P02W14_ArcEnd   := [[0,0,0],[1,0,0,0],[0,0,0,0],[9E9,9E9,9E9,9E9,9E9,9E9]];
    PERS robtarget P02W14_Approach := [[0,0,0],[1,0,0,0],[0,0,0,0],[9E9,9E9,9E9,9E9,9E9,9E9]];
    PERS robtarget P02W14_Retract  := [[0,0,0],[1,0,0,0],[0,0,0,0],[9E9,9E9,9E9,9E9,9E9,9E9]];
    PERS robtarget P02W14_Trans    := [[0,0,0],[1,0,0,0],[0,0,0,0],[9E9,9E9,9E9,9E9,9E9,9E9]];
    PERS bool P02W15_Used := FALSE;
    PERS num  P02W15_SubType := 0;
    PERS num  P02W15_ToolSel := 0;
    PERS num  P02W15_LenMM := 0;
    PERS robtarget P02W15_ArcStart := [[0,0,0],[1,0,0,0],[0,0,0,0],[9E9,9E9,9E9,9E9,9E9,9E9]];
    PERS robtarget P02W15_ArcEnd   := [[0,0,0],[1,0,0,0],[0,0,0,0],[9E9,9E9,9E9,9E9,9E9,9E9]];
    PERS robtarget P02W15_Approach := [[0,0,0],[1,0,0,0],[0,0,0,0],[9E9,9E9,9E9,9E9,9E9,9E9]];
    PERS robtarget P02W15_Retract  := [[0,0,0],[1,0,0,0],[0,0,0,0],[9E9,9E9,9E9,9E9,9E9,9E9]];
    PERS robtarget P02W15_Trans    := [[0,0,0],[1,0,0,0],[0,0,0,0],[9E9,9E9,9E9,9E9,9E9,9E9]];
    PERS bool P02W16_Used := FALSE;
    PERS num  P02W16_SubType := 0;
    PERS num  P02W16_ToolSel := 0;
    PERS num  P02W16_LenMM := 0;
    PERS robtarget P02W16_ArcStart := [[0,0,0],[1,0,0,0],[0,0,0,0],[9E9,9E9,9E9,9E9,9E9,9E9]];
    PERS robtarget P02W16_ArcEnd   := [[0,0,0],[1,0,0,0],[0,0,0,0],[9E9,9E9,9E9,9E9,9E9,9E9]];
    PERS robtarget P02W16_Approach := [[0,0,0],[1,0,0,0],[0,0,0,0],[9E9,9E9,9E9,9E9,9E9,9E9]];
    PERS robtarget P02W16_Retract  := [[0,0,0],[1,0,0,0],[0,0,0,0],[9E9,9E9,9E9,9E9,9E9,9E9]];
    PERS robtarget P02W16_Trans    := [[0,0,0],[1,0,0,0],[0,0,0,0],[9E9,9E9,9E9,9E9,9E9,9E9]];
    PERS bool P02W17_Used := FALSE;
    PERS num  P02W17_SubType := 0;
    PERS num  P02W17_ToolSel := 0;
    PERS num  P02W17_LenMM := 0;
    PERS robtarget P02W17_ArcStart := [[0,0,0],[1,0,0,0],[0,0,0,0],[9E9,9E9,9E9,9E9,9E9,9E9]];
    PERS robtarget P02W17_ArcEnd   := [[0,0,0],[1,0,0,0],[0,0,0,0],[9E9,9E9,9E9,9E9,9E9,9E9]];
    PERS robtarget P02W17_Approach := [[0,0,0],[1,0,0,0],[0,0,0,0],[9E9,9E9,9E9,9E9,9E9,9E9]];
    PERS robtarget P02W17_Retract  := [[0,0,0],[1,0,0,0],[0,0,0,0],[9E9,9E9,9E9,9E9,9E9,9E9]];
    PERS robtarget P02W17_Trans    := [[0,0,0],[1,0,0,0],[0,0,0,0],[9E9,9E9,9E9,9E9,9E9,9E9]];
    PERS bool P02W18_Used := FALSE;
    PERS num  P02W18_SubType := 0;
    PERS num  P02W18_ToolSel := 0;
    PERS num  P02W18_LenMM := 0;
    PERS robtarget P02W18_ArcStart := [[0,0,0],[1,0,0,0],[0,0,0,0],[9E9,9E9,9E9,9E9,9E9,9E9]];
    PERS robtarget P02W18_ArcEnd   := [[0,0,0],[1,0,0,0],[0,0,0,0],[9E9,9E9,9E9,9E9,9E9,9E9]];
    PERS robtarget P02W18_Approach := [[0,0,0],[1,0,0,0],[0,0,0,0],[9E9,9E9,9E9,9E9,9E9,9E9]];
    PERS robtarget P02W18_Retract  := [[0,0,0],[1,0,0,0],[0,0,0,0],[9E9,9E9,9E9,9E9,9E9,9E9]];
    PERS robtarget P02W18_Trans    := [[0,0,0],[1,0,0,0],[0,0,0,0],[9E9,9E9,9E9,9E9,9E9,9E9]];
    PERS bool P02W19_Used := FALSE;
    PERS num  P02W19_SubType := 0;
    PERS num  P02W19_ToolSel := 0;
    PERS num  P02W19_LenMM := 0;
    PERS robtarget P02W19_ArcStart := [[0,0,0],[1,0,0,0],[0,0,0,0],[9E9,9E9,9E9,9E9,9E9,9E9]];
    PERS robtarget P02W19_ArcEnd   := [[0,0,0],[1,0,0,0],[0,0,0,0],[9E9,9E9,9E9,9E9,9E9,9E9]];
    PERS robtarget P02W19_Approach := [[0,0,0],[1,0,0,0],[0,0,0,0],[9E9,9E9,9E9,9E9,9E9,9E9]];
    PERS robtarget P02W19_Retract  := [[0,0,0],[1,0,0,0],[0,0,0,0],[9E9,9E9,9E9,9E9,9E9,9E9]];
    PERS robtarget P02W19_Trans    := [[0,0,0],[1,0,0,0],[0,0,0,0],[9E9,9E9,9E9,9E9,9E9,9E9]];
    PERS bool P02W20_Used := FALSE;
    PERS num  P02W20_SubType := 0;
    PERS num  P02W20_ToolSel := 0;
    PERS num  P02W20_LenMM := 0;
    PERS robtarget P02W20_ArcStart := [[0,0,0],[1,0,0,0],[0,0,0,0],[9E9,9E9,9E9,9E9,9E9,9E9]];
    PERS robtarget P02W20_ArcEnd   := [[0,0,0],[1,0,0,0],[0,0,0,0],[9E9,9E9,9E9,9E9,9E9,9E9]];
    PERS robtarget P02W20_Approach := [[0,0,0],[1,0,0,0],[0,0,0,0],[9E9,9E9,9E9,9E9,9E9,9E9]];
    PERS robtarget P02W20_Retract  := [[0,0,0],[1,0,0,0],[0,0,0,0],[9E9,9E9,9E9,9E9,9E9,9E9]];
    PERS robtarget P02W20_Trans    := [[0,0,0],[1,0,0,0],[0,0,0,0],[9E9,9E9,9E9,9E9,9E9,9E9]];
    PERS bool P02W21_Used := FALSE;
    PERS num  P02W21_SubType := 0;
    PERS num  P02W21_ToolSel := 0;
    PERS num  P02W21_LenMM := 0;
    PERS robtarget P02W21_ArcStart := [[0,0,0],[1,0,0,0],[0,0,0,0],[9E9,9E9,9E9,9E9,9E9,9E9]];
    PERS robtarget P02W21_ArcEnd   := [[0,0,0],[1,0,0,0],[0,0,0,0],[9E9,9E9,9E9,9E9,9E9,9E9]];
    PERS robtarget P02W21_Approach := [[0,0,0],[1,0,0,0],[0,0,0,0],[9E9,9E9,9E9,9E9,9E9,9E9]];
    PERS robtarget P02W21_Retract  := [[0,0,0],[1,0,0,0],[0,0,0,0],[9E9,9E9,9E9,9E9,9E9,9E9]];
    PERS robtarget P02W21_Trans    := [[0,0,0],[1,0,0,0],[0,0,0,0],[9E9,9E9,9E9,9E9,9E9,9E9]];
    PERS bool P02W22_Used := FALSE;
    PERS num  P02W22_SubType := 0;
    PERS num  P02W22_ToolSel := 0;
    PERS num  P02W22_LenMM := 0;
    PERS robtarget P02W22_ArcStart := [[0,0,0],[1,0,0,0],[0,0,0,0],[9E9,9E9,9E9,9E9,9E9,9E9]];
    PERS robtarget P02W22_ArcEnd   := [[0,0,0],[1,0,0,0],[0,0,0,0],[9E9,9E9,9E9,9E9,9E9,9E9]];
    PERS robtarget P02W22_Approach := [[0,0,0],[1,0,0,0],[0,0,0,0],[9E9,9E9,9E9,9E9,9E9,9E9]];
    PERS robtarget P02W22_Retract  := [[0,0,0],[1,0,0,0],[0,0,0,0],[9E9,9E9,9E9,9E9,9E9,9E9]];
    PERS robtarget P02W22_Trans    := [[0,0,0],[1,0,0,0],[0,0,0,0],[9E9,9E9,9E9,9E9,9E9,9E9]];
    PERS bool P02W23_Used := FALSE;
    PERS num  P02W23_SubType := 0;
    PERS num  P02W23_ToolSel := 0;
    PERS num  P02W23_LenMM := 0;
    PERS robtarget P02W23_ArcStart := [[0,0,0],[1,0,0,0],[0,0,0,0],[9E9,9E9,9E9,9E9,9E9,9E9]];
    PERS robtarget P02W23_ArcEnd   := [[0,0,0],[1,0,0,0],[0,0,0,0],[9E9,9E9,9E9,9E9,9E9,9E9]];
    PERS robtarget P02W23_Approach := [[0,0,0],[1,0,0,0],[0,0,0,0],[9E9,9E9,9E9,9E9,9E9,9E9]];
    PERS robtarget P02W23_Retract  := [[0,0,0],[1,0,0,0],[0,0,0,0],[9E9,9E9,9E9,9E9,9E9,9E9]];
    PERS robtarget P02W23_Trans    := [[0,0,0],[1,0,0,0],[0,0,0,0],[9E9,9E9,9E9,9E9,9E9,9E9]];
    PERS bool P02W24_Used := FALSE;
    PERS num  P02W24_SubType := 0;
    PERS num  P02W24_ToolSel := 0;
    PERS num  P02W24_LenMM := 0;
    PERS robtarget P02W24_ArcStart := [[0,0,0],[1,0,0,0],[0,0,0,0],[9E9,9E9,9E9,9E9,9E9,9E9]];
    PERS robtarget P02W24_ArcEnd   := [[0,0,0],[1,0,0,0],[0,0,0,0],[9E9,9E9,9E9,9E9,9E9,9E9]];
    PERS robtarget P02W24_Approach := [[0,0,0],[1,0,0,0],[0,0,0,0],[9E9,9E9,9E9,9E9,9E9,9E9]];
    PERS robtarget P02W24_Retract  := [[0,0,0],[1,0,0,0],[0,0,0,0],[9E9,9E9,9E9,9E9,9E9,9E9]];
    PERS robtarget P02W24_Trans    := [[0,0,0],[1,0,0,0],[0,0,0,0],[9E9,9E9,9E9,9E9,9E9,9E9]];
    PERS bool P02W25_Used := FALSE;
    PERS num  P02W25_SubType := 0;
    PERS num  P02W25_ToolSel := 0;
    PERS num  P02W25_LenMM := 0;
    PERS robtarget P02W25_ArcStart := [[0,0,0],[1,0,0,0],[0,0,0,0],[9E9,9E9,9E9,9E9,9E9,9E9]];
    PERS robtarget P02W25_ArcEnd   := [[0,0,0],[1,0,0,0],[0,0,0,0],[9E9,9E9,9E9,9E9,9E9,9E9]];
    PERS robtarget P02W25_Approach := [[0,0,0],[1,0,0,0],[0,0,0,0],[9E9,9E9,9E9,9E9,9E9,9E9]];
    PERS robtarget P02W25_Retract  := [[0,0,0],[1,0,0,0],[0,0,0,0],[9E9,9E9,9E9,9E9,9E9,9E9]];
    PERS robtarget P02W25_Trans    := [[0,0,0],[1,0,0,0],[0,0,0,0],[9E9,9E9,9E9,9E9,9E9,9E9]];
    PERS bool P02W26_Used := FALSE;
    PERS num  P02W26_SubType := 0;
    PERS num  P02W26_ToolSel := 0;
    PERS num  P02W26_LenMM := 0;
    PERS robtarget P02W26_ArcStart := [[0,0,0],[1,0,0,0],[0,0,0,0],[9E9,9E9,9E9,9E9,9E9,9E9]];
    PERS robtarget P02W26_ArcEnd   := [[0,0,0],[1,0,0,0],[0,0,0,0],[9E9,9E9,9E9,9E9,9E9,9E9]];
    PERS robtarget P02W26_Approach := [[0,0,0],[1,0,0,0],[0,0,0,0],[9E9,9E9,9E9,9E9,9E9,9E9]];
    PERS robtarget P02W26_Retract  := [[0,0,0],[1,0,0,0],[0,0,0,0],[9E9,9E9,9E9,9E9,9E9,9E9]];
    PERS robtarget P02W26_Trans    := [[0,0,0],[1,0,0,0],[0,0,0,0],[9E9,9E9,9E9,9E9,9E9,9E9]];
    PERS bool P02W27_Used := FALSE;
    PERS num  P02W27_SubType := 0;
    PERS num  P02W27_ToolSel := 0;
    PERS num  P02W27_LenMM := 0;
    PERS robtarget P02W27_ArcStart := [[0,0,0],[1,0,0,0],[0,0,0,0],[9E9,9E9,9E9,9E9,9E9,9E9]];
    PERS robtarget P02W27_ArcEnd   := [[0,0,0],[1,0,0,0],[0,0,0,0],[9E9,9E9,9E9,9E9,9E9,9E9]];
    PERS robtarget P02W27_Approach := [[0,0,0],[1,0,0,0],[0,0,0,0],[9E9,9E9,9E9,9E9,9E9,9E9]];
    PERS robtarget P02W27_Retract  := [[0,0,0],[1,0,0,0],[0,0,0,0],[9E9,9E9,9E9,9E9,9E9,9E9]];
    PERS robtarget P02W27_Trans    := [[0,0,0],[1,0,0,0],[0,0,0,0],[9E9,9E9,9E9,9E9,9E9,9E9]];
    PERS bool P02W28_Used := FALSE;
    PERS num  P02W28_SubType := 0;
    PERS num  P02W28_ToolSel := 0;
    PERS num  P02W28_LenMM := 0;
    PERS robtarget P02W28_ArcStart := [[0,0,0],[1,0,0,0],[0,0,0,0],[9E9,9E9,9E9,9E9,9E9,9E9]];
    PERS robtarget P02W28_ArcEnd   := [[0,0,0],[1,0,0,0],[0,0,0,0],[9E9,9E9,9E9,9E9,9E9,9E9]];
    PERS robtarget P02W28_Approach := [[0,0,0],[1,0,0,0],[0,0,0,0],[9E9,9E9,9E9,9E9,9E9,9E9]];
    PERS robtarget P02W28_Retract  := [[0,0,0],[1,0,0,0],[0,0,0,0],[9E9,9E9,9E9,9E9,9E9,9E9]];
    PERS robtarget P02W28_Trans    := [[0,0,0],[1,0,0,0],[0,0,0,0],[9E9,9E9,9E9,9E9,9E9,9E9]];
    PERS bool P02W29_Used := FALSE;
    PERS num  P02W29_SubType := 0;
    PERS num  P02W29_ToolSel := 0;
    PERS num  P02W29_LenMM := 0;
    PERS robtarget P02W29_ArcStart := [[0,0,0],[1,0,0,0],[0,0,0,0],[9E9,9E9,9E9,9E9,9E9,9E9]];
    PERS robtarget P02W29_ArcEnd   := [[0,0,0],[1,0,0,0],[0,0,0,0],[9E9,9E9,9E9,9E9,9E9,9E9]];
    PERS robtarget P02W29_Approach := [[0,0,0],[1,0,0,0],[0,0,0,0],[9E9,9E9,9E9,9E9,9E9,9E9]];
    PERS robtarget P02W29_Retract  := [[0,0,0],[1,0,0,0],[0,0,0,0],[9E9,9E9,9E9,9E9,9E9,9E9]];
    PERS robtarget P02W29_Trans    := [[0,0,0],[1,0,0,0],[0,0,0,0],[9E9,9E9,9E9,9E9,9E9,9E9]];
    PERS bool P02W30_Used := FALSE;
    PERS num  P02W30_SubType := 0;
    PERS num  P02W30_ToolSel := 0;
    PERS num  P02W30_LenMM := 0;
    PERS robtarget P02W30_ArcStart := [[0,0,0],[1,0,0,0],[0,0,0,0],[9E9,9E9,9E9,9E9,9E9,9E9]];
    PERS robtarget P02W30_ArcEnd   := [[0,0,0],[1,0,0,0],[0,0,0,0],[9E9,9E9,9E9,9E9,9E9,9E9]];
    PERS robtarget P02W30_Approach := [[0,0,0],[1,0,0,0],[0,0,0,0],[9E9,9E9,9E9,9E9,9E9,9E9]];
    PERS robtarget P02W30_Retract  := [[0,0,0],[1,0,0,0],[0,0,0,0],[9E9,9E9,9E9,9E9,9E9,9E9]];
    PERS robtarget P02W30_Trans    := [[0,0,0],[1,0,0,0],[0,0,0,0],[9E9,9E9,9E9,9E9,9E9,9E9]];

    ! ---- P03 weld slots ----
    PERS bool P03W01_Used := FALSE;
    PERS num  P03W01_SubType := 0;
    PERS num  P03W01_ToolSel := 0;
    PERS num  P03W01_LenMM := 0;
    PERS robtarget P03W01_ArcStart := [[0,0,0],[1,0,0,0],[0,0,0,0],[9E9,9E9,9E9,9E9,9E9,9E9]];
    PERS robtarget P03W01_ArcEnd   := [[0,0,0],[1,0,0,0],[0,0,0,0],[9E9,9E9,9E9,9E9,9E9,9E9]];
    PERS robtarget P03W01_Approach := [[0,0,0],[1,0,0,0],[0,0,0,0],[9E9,9E9,9E9,9E9,9E9,9E9]];
    PERS robtarget P03W01_Retract  := [[0,0,0],[1,0,0,0],[0,0,0,0],[9E9,9E9,9E9,9E9,9E9,9E9]];
    PERS robtarget P03W01_Trans    := [[0,0,0],[1,0,0,0],[0,0,0,0],[9E9,9E9,9E9,9E9,9E9,9E9]];
    PERS bool P03W02_Used := FALSE;
    PERS num  P03W02_SubType := 0;
    PERS num  P03W02_ToolSel := 0;
    PERS num  P03W02_LenMM := 0;
    PERS robtarget P03W02_ArcStart := [[0,0,0],[1,0,0,0],[0,0,0,0],[9E9,9E9,9E9,9E9,9E9,9E9]];
    PERS robtarget P03W02_ArcEnd   := [[0,0,0],[1,0,0,0],[0,0,0,0],[9E9,9E9,9E9,9E9,9E9,9E9]];
    PERS robtarget P03W02_Approach := [[0,0,0],[1,0,0,0],[0,0,0,0],[9E9,9E9,9E9,9E9,9E9,9E9]];
    PERS robtarget P03W02_Retract  := [[0,0,0],[1,0,0,0],[0,0,0,0],[9E9,9E9,9E9,9E9,9E9,9E9]];
    PERS robtarget P03W02_Trans    := [[0,0,0],[1,0,0,0],[0,0,0,0],[9E9,9E9,9E9,9E9,9E9,9E9]];
    PERS bool P03W03_Used := FALSE;
    PERS num  P03W03_SubType := 0;
    PERS num  P03W03_ToolSel := 0;
    PERS num  P03W03_LenMM := 0;
    PERS robtarget P03W03_ArcStart := [[0,0,0],[1,0,0,0],[0,0,0,0],[9E9,9E9,9E9,9E9,9E9,9E9]];
    PERS robtarget P03W03_ArcEnd   := [[0,0,0],[1,0,0,0],[0,0,0,0],[9E9,9E9,9E9,9E9,9E9,9E9]];
    PERS robtarget P03W03_Approach := [[0,0,0],[1,0,0,0],[0,0,0,0],[9E9,9E9,9E9,9E9,9E9,9E9]];
    PERS robtarget P03W03_Retract  := [[0,0,0],[1,0,0,0],[0,0,0,0],[9E9,9E9,9E9,9E9,9E9,9E9]];
    PERS robtarget P03W03_Trans    := [[0,0,0],[1,0,0,0],[0,0,0,0],[9E9,9E9,9E9,9E9,9E9,9E9]];
    PERS bool P03W04_Used := FALSE;
    PERS num  P03W04_SubType := 0;
    PERS num  P03W04_ToolSel := 0;
    PERS num  P03W04_LenMM := 0;
    PERS robtarget P03W04_ArcStart := [[0,0,0],[1,0,0,0],[0,0,0,0],[9E9,9E9,9E9,9E9,9E9,9E9]];
    PERS robtarget P03W04_ArcEnd   := [[0,0,0],[1,0,0,0],[0,0,0,0],[9E9,9E9,9E9,9E9,9E9,9E9]];
    PERS robtarget P03W04_Approach := [[0,0,0],[1,0,0,0],[0,0,0,0],[9E9,9E9,9E9,9E9,9E9,9E9]];
    PERS robtarget P03W04_Retract  := [[0,0,0],[1,0,0,0],[0,0,0,0],[9E9,9E9,9E9,9E9,9E9,9E9]];
    PERS robtarget P03W04_Trans    := [[0,0,0],[1,0,0,0],[0,0,0,0],[9E9,9E9,9E9,9E9,9E9,9E9]];
    PERS bool P03W05_Used := FALSE;
    PERS num  P03W05_SubType := 0;
    PERS num  P03W05_ToolSel := 0;
    PERS num  P03W05_LenMM := 0;
    PERS robtarget P03W05_ArcStart := [[0,0,0],[1,0,0,0],[0,0,0,0],[9E9,9E9,9E9,9E9,9E9,9E9]];
    PERS robtarget P03W05_ArcEnd   := [[0,0,0],[1,0,0,0],[0,0,0,0],[9E9,9E9,9E9,9E9,9E9,9E9]];
    PERS robtarget P03W05_Approach := [[0,0,0],[1,0,0,0],[0,0,0,0],[9E9,9E9,9E9,9E9,9E9,9E9]];
    PERS robtarget P03W05_Retract  := [[0,0,0],[1,0,0,0],[0,0,0,0],[9E9,9E9,9E9,9E9,9E9,9E9]];
    PERS robtarget P03W05_Trans    := [[0,0,0],[1,0,0,0],[0,0,0,0],[9E9,9E9,9E9,9E9,9E9,9E9]];
    PERS bool P03W06_Used := FALSE;
    PERS num  P03W06_SubType := 0;
    PERS num  P03W06_ToolSel := 0;
    PERS num  P03W06_LenMM := 0;
    PERS robtarget P03W06_ArcStart := [[0,0,0],[1,0,0,0],[0,0,0,0],[9E9,9E9,9E9,9E9,9E9,9E9]];
    PERS robtarget P03W06_ArcEnd   := [[0,0,0],[1,0,0,0],[0,0,0,0],[9E9,9E9,9E9,9E9,9E9,9E9]];
    PERS robtarget P03W06_Approach := [[0,0,0],[1,0,0,0],[0,0,0,0],[9E9,9E9,9E9,9E9,9E9,9E9]];
    PERS robtarget P03W06_Retract  := [[0,0,0],[1,0,0,0],[0,0,0,0],[9E9,9E9,9E9,9E9,9E9,9E9]];
    PERS robtarget P03W06_Trans    := [[0,0,0],[1,0,0,0],[0,0,0,0],[9E9,9E9,9E9,9E9,9E9,9E9]];
    PERS bool P03W07_Used := FALSE;
    PERS num  P03W07_SubType := 0;
    PERS num  P03W07_ToolSel := 0;
    PERS num  P03W07_LenMM := 0;
    PERS robtarget P03W07_ArcStart := [[0,0,0],[1,0,0,0],[0,0,0,0],[9E9,9E9,9E9,9E9,9E9,9E9]];
    PERS robtarget P03W07_ArcEnd   := [[0,0,0],[1,0,0,0],[0,0,0,0],[9E9,9E9,9E9,9E9,9E9,9E9]];
    PERS robtarget P03W07_Approach := [[0,0,0],[1,0,0,0],[0,0,0,0],[9E9,9E9,9E9,9E9,9E9,9E9]];
    PERS robtarget P03W07_Retract  := [[0,0,0],[1,0,0,0],[0,0,0,0],[9E9,9E9,9E9,9E9,9E9,9E9]];
    PERS robtarget P03W07_Trans    := [[0,0,0],[1,0,0,0],[0,0,0,0],[9E9,9E9,9E9,9E9,9E9,9E9]];
    PERS bool P03W08_Used := FALSE;
    PERS num  P03W08_SubType := 0;
    PERS num  P03W08_ToolSel := 0;
    PERS num  P03W08_LenMM := 0;
    PERS robtarget P03W08_ArcStart := [[0,0,0],[1,0,0,0],[0,0,0,0],[9E9,9E9,9E9,9E9,9E9,9E9]];
    PERS robtarget P03W08_ArcEnd   := [[0,0,0],[1,0,0,0],[0,0,0,0],[9E9,9E9,9E9,9E9,9E9,9E9]];
    PERS robtarget P03W08_Approach := [[0,0,0],[1,0,0,0],[0,0,0,0],[9E9,9E9,9E9,9E9,9E9,9E9]];
    PERS robtarget P03W08_Retract  := [[0,0,0],[1,0,0,0],[0,0,0,0],[9E9,9E9,9E9,9E9,9E9,9E9]];
    PERS robtarget P03W08_Trans    := [[0,0,0],[1,0,0,0],[0,0,0,0],[9E9,9E9,9E9,9E9,9E9,9E9]];
    PERS bool P03W09_Used := FALSE;
    PERS num  P03W09_SubType := 0;
    PERS num  P03W09_ToolSel := 0;
    PERS num  P03W09_LenMM := 0;
    PERS robtarget P03W09_ArcStart := [[0,0,0],[1,0,0,0],[0,0,0,0],[9E9,9E9,9E9,9E9,9E9,9E9]];
    PERS robtarget P03W09_ArcEnd   := [[0,0,0],[1,0,0,0],[0,0,0,0],[9E9,9E9,9E9,9E9,9E9,9E9]];
    PERS robtarget P03W09_Approach := [[0,0,0],[1,0,0,0],[0,0,0,0],[9E9,9E9,9E9,9E9,9E9,9E9]];
    PERS robtarget P03W09_Retract  := [[0,0,0],[1,0,0,0],[0,0,0,0],[9E9,9E9,9E9,9E9,9E9,9E9]];
    PERS robtarget P03W09_Trans    := [[0,0,0],[1,0,0,0],[0,0,0,0],[9E9,9E9,9E9,9E9,9E9,9E9]];
    PERS bool P03W10_Used := FALSE;
    PERS num  P03W10_SubType := 0;
    PERS num  P03W10_ToolSel := 0;
    PERS num  P03W10_LenMM := 0;
    PERS robtarget P03W10_ArcStart := [[0,0,0],[1,0,0,0],[0,0,0,0],[9E9,9E9,9E9,9E9,9E9,9E9]];
    PERS robtarget P03W10_ArcEnd   := [[0,0,0],[1,0,0,0],[0,0,0,0],[9E9,9E9,9E9,9E9,9E9,9E9]];
    PERS robtarget P03W10_Approach := [[0,0,0],[1,0,0,0],[0,0,0,0],[9E9,9E9,9E9,9E9,9E9,9E9]];
    PERS robtarget P03W10_Retract  := [[0,0,0],[1,0,0,0],[0,0,0,0],[9E9,9E9,9E9,9E9,9E9,9E9]];
    PERS robtarget P03W10_Trans    := [[0,0,0],[1,0,0,0],[0,0,0,0],[9E9,9E9,9E9,9E9,9E9,9E9]];
    PERS bool P03W11_Used := FALSE;
    PERS num  P03W11_SubType := 0;
    PERS num  P03W11_ToolSel := 0;
    PERS num  P03W11_LenMM := 0;
    PERS robtarget P03W11_ArcStart := [[0,0,0],[1,0,0,0],[0,0,0,0],[9E9,9E9,9E9,9E9,9E9,9E9]];
    PERS robtarget P03W11_ArcEnd   := [[0,0,0],[1,0,0,0],[0,0,0,0],[9E9,9E9,9E9,9E9,9E9,9E9]];
    PERS robtarget P03W11_Approach := [[0,0,0],[1,0,0,0],[0,0,0,0],[9E9,9E9,9E9,9E9,9E9,9E9]];
    PERS robtarget P03W11_Retract  := [[0,0,0],[1,0,0,0],[0,0,0,0],[9E9,9E9,9E9,9E9,9E9,9E9]];
    PERS robtarget P03W11_Trans    := [[0,0,0],[1,0,0,0],[0,0,0,0],[9E9,9E9,9E9,9E9,9E9,9E9]];
    PERS bool P03W12_Used := FALSE;
    PERS num  P03W12_SubType := 0;
    PERS num  P03W12_ToolSel := 0;
    PERS num  P03W12_LenMM := 0;
    PERS robtarget P03W12_ArcStart := [[0,0,0],[1,0,0,0],[0,0,0,0],[9E9,9E9,9E9,9E9,9E9,9E9]];
    PERS robtarget P03W12_ArcEnd   := [[0,0,0],[1,0,0,0],[0,0,0,0],[9E9,9E9,9E9,9E9,9E9,9E9]];
    PERS robtarget P03W12_Approach := [[0,0,0],[1,0,0,0],[0,0,0,0],[9E9,9E9,9E9,9E9,9E9,9E9]];
    PERS robtarget P03W12_Retract  := [[0,0,0],[1,0,0,0],[0,0,0,0],[9E9,9E9,9E9,9E9,9E9,9E9]];
    PERS robtarget P03W12_Trans    := [[0,0,0],[1,0,0,0],[0,0,0,0],[9E9,9E9,9E9,9E9,9E9,9E9]];
    PERS bool P03W13_Used := FALSE;
    PERS num  P03W13_SubType := 0;
    PERS num  P03W13_ToolSel := 0;
    PERS num  P03W13_LenMM := 0;
    PERS robtarget P03W13_ArcStart := [[0,0,0],[1,0,0,0],[0,0,0,0],[9E9,9E9,9E9,9E9,9E9,9E9]];
    PERS robtarget P03W13_ArcEnd   := [[0,0,0],[1,0,0,0],[0,0,0,0],[9E9,9E9,9E9,9E9,9E9,9E9]];
    PERS robtarget P03W13_Approach := [[0,0,0],[1,0,0,0],[0,0,0,0],[9E9,9E9,9E9,9E9,9E9,9E9]];
    PERS robtarget P03W13_Retract  := [[0,0,0],[1,0,0,0],[0,0,0,0],[9E9,9E9,9E9,9E9,9E9,9E9]];
    PERS robtarget P03W13_Trans    := [[0,0,0],[1,0,0,0],[0,0,0,0],[9E9,9E9,9E9,9E9,9E9,9E9]];
    PERS bool P03W14_Used := FALSE;
    PERS num  P03W14_SubType := 0;
    PERS num  P03W14_ToolSel := 0;
    PERS num  P03W14_LenMM := 0;
    PERS robtarget P03W14_ArcStart := [[0,0,0],[1,0,0,0],[0,0,0,0],[9E9,9E9,9E9,9E9,9E9,9E9]];
    PERS robtarget P03W14_ArcEnd   := [[0,0,0],[1,0,0,0],[0,0,0,0],[9E9,9E9,9E9,9E9,9E9,9E9]];
    PERS robtarget P03W14_Approach := [[0,0,0],[1,0,0,0],[0,0,0,0],[9E9,9E9,9E9,9E9,9E9,9E9]];
    PERS robtarget P03W14_Retract  := [[0,0,0],[1,0,0,0],[0,0,0,0],[9E9,9E9,9E9,9E9,9E9,9E9]];
    PERS robtarget P03W14_Trans    := [[0,0,0],[1,0,0,0],[0,0,0,0],[9E9,9E9,9E9,9E9,9E9,9E9]];
    PERS bool P03W15_Used := FALSE;
    PERS num  P03W15_SubType := 0;
    PERS num  P03W15_ToolSel := 0;
    PERS num  P03W15_LenMM := 0;
    PERS robtarget P03W15_ArcStart := [[0,0,0],[1,0,0,0],[0,0,0,0],[9E9,9E9,9E9,9E9,9E9,9E9]];
    PERS robtarget P03W15_ArcEnd   := [[0,0,0],[1,0,0,0],[0,0,0,0],[9E9,9E9,9E9,9E9,9E9,9E9]];
    PERS robtarget P03W15_Approach := [[0,0,0],[1,0,0,0],[0,0,0,0],[9E9,9E9,9E9,9E9,9E9,9E9]];
    PERS robtarget P03W15_Retract  := [[0,0,0],[1,0,0,0],[0,0,0,0],[9E9,9E9,9E9,9E9,9E9,9E9]];
    PERS robtarget P03W15_Trans    := [[0,0,0],[1,0,0,0],[0,0,0,0],[9E9,9E9,9E9,9E9,9E9,9E9]];
    PERS bool P03W16_Used := FALSE;
    PERS num  P03W16_SubType := 0;
    PERS num  P03W16_ToolSel := 0;
    PERS num  P03W16_LenMM := 0;
    PERS robtarget P03W16_ArcStart := [[0,0,0],[1,0,0,0],[0,0,0,0],[9E9,9E9,9E9,9E9,9E9,9E9]];
    PERS robtarget P03W16_ArcEnd   := [[0,0,0],[1,0,0,0],[0,0,0,0],[9E9,9E9,9E9,9E9,9E9,9E9]];
    PERS robtarget P03W16_Approach := [[0,0,0],[1,0,0,0],[0,0,0,0],[9E9,9E9,9E9,9E9,9E9,9E9]];
    PERS robtarget P03W16_Retract  := [[0,0,0],[1,0,0,0],[0,0,0,0],[9E9,9E9,9E9,9E9,9E9,9E9]];
    PERS robtarget P03W16_Trans    := [[0,0,0],[1,0,0,0],[0,0,0,0],[9E9,9E9,9E9,9E9,9E9,9E9]];
    PERS bool P03W17_Used := FALSE;
    PERS num  P03W17_SubType := 0;
    PERS num  P03W17_ToolSel := 0;
    PERS num  P03W17_LenMM := 0;
    PERS robtarget P03W17_ArcStart := [[0,0,0],[1,0,0,0],[0,0,0,0],[9E9,9E9,9E9,9E9,9E9,9E9]];
    PERS robtarget P03W17_ArcEnd   := [[0,0,0],[1,0,0,0],[0,0,0,0],[9E9,9E9,9E9,9E9,9E9,9E9]];
    PERS robtarget P03W17_Approach := [[0,0,0],[1,0,0,0],[0,0,0,0],[9E9,9E9,9E9,9E9,9E9,9E9]];
    PERS robtarget P03W17_Retract  := [[0,0,0],[1,0,0,0],[0,0,0,0],[9E9,9E9,9E9,9E9,9E9,9E9]];
    PERS robtarget P03W17_Trans    := [[0,0,0],[1,0,0,0],[0,0,0,0],[9E9,9E9,9E9,9E9,9E9,9E9]];
    PERS bool P03W18_Used := FALSE;
    PERS num  P03W18_SubType := 0;
    PERS num  P03W18_ToolSel := 0;
    PERS num  P03W18_LenMM := 0;
    PERS robtarget P03W18_ArcStart := [[0,0,0],[1,0,0,0],[0,0,0,0],[9E9,9E9,9E9,9E9,9E9,9E9]];
    PERS robtarget P03W18_ArcEnd   := [[0,0,0],[1,0,0,0],[0,0,0,0],[9E9,9E9,9E9,9E9,9E9,9E9]];
    PERS robtarget P03W18_Approach := [[0,0,0],[1,0,0,0],[0,0,0,0],[9E9,9E9,9E9,9E9,9E9,9E9]];
    PERS robtarget P03W18_Retract  := [[0,0,0],[1,0,0,0],[0,0,0,0],[9E9,9E9,9E9,9E9,9E9,9E9]];
    PERS robtarget P03W18_Trans    := [[0,0,0],[1,0,0,0],[0,0,0,0],[9E9,9E9,9E9,9E9,9E9,9E9]];
    PERS bool P03W19_Used := FALSE;
    PERS num  P03W19_SubType := 0;
    PERS num  P03W19_ToolSel := 0;
    PERS num  P03W19_LenMM := 0;
    PERS robtarget P03W19_ArcStart := [[0,0,0],[1,0,0,0],[0,0,0,0],[9E9,9E9,9E9,9E9,9E9,9E9]];
    PERS robtarget P03W19_ArcEnd   := [[0,0,0],[1,0,0,0],[0,0,0,0],[9E9,9E9,9E9,9E9,9E9,9E9]];
    PERS robtarget P03W19_Approach := [[0,0,0],[1,0,0,0],[0,0,0,0],[9E9,9E9,9E9,9E9,9E9,9E9]];
    PERS robtarget P03W19_Retract  := [[0,0,0],[1,0,0,0],[0,0,0,0],[9E9,9E9,9E9,9E9,9E9,9E9]];
    PERS robtarget P03W19_Trans    := [[0,0,0],[1,0,0,0],[0,0,0,0],[9E9,9E9,9E9,9E9,9E9,9E9]];
    PERS bool P03W20_Used := FALSE;
    PERS num  P03W20_SubType := 0;
    PERS num  P03W20_ToolSel := 0;
    PERS num  P03W20_LenMM := 0;
    PERS robtarget P03W20_ArcStart := [[0,0,0],[1,0,0,0],[0,0,0,0],[9E9,9E9,9E9,9E9,9E9,9E9]];
    PERS robtarget P03W20_ArcEnd   := [[0,0,0],[1,0,0,0],[0,0,0,0],[9E9,9E9,9E9,9E9,9E9,9E9]];
    PERS robtarget P03W20_Approach := [[0,0,0],[1,0,0,0],[0,0,0,0],[9E9,9E9,9E9,9E9,9E9,9E9]];
    PERS robtarget P03W20_Retract  := [[0,0,0],[1,0,0,0],[0,0,0,0],[9E9,9E9,9E9,9E9,9E9,9E9]];
    PERS robtarget P03W20_Trans    := [[0,0,0],[1,0,0,0],[0,0,0,0],[9E9,9E9,9E9,9E9,9E9,9E9]];
    PERS bool P03W21_Used := FALSE;
    PERS num  P03W21_SubType := 0;
    PERS num  P03W21_ToolSel := 0;
    PERS num  P03W21_LenMM := 0;
    PERS robtarget P03W21_ArcStart := [[0,0,0],[1,0,0,0],[0,0,0,0],[9E9,9E9,9E9,9E9,9E9,9E9]];
    PERS robtarget P03W21_ArcEnd   := [[0,0,0],[1,0,0,0],[0,0,0,0],[9E9,9E9,9E9,9E9,9E9,9E9]];
    PERS robtarget P03W21_Approach := [[0,0,0],[1,0,0,0],[0,0,0,0],[9E9,9E9,9E9,9E9,9E9,9E9]];
    PERS robtarget P03W21_Retract  := [[0,0,0],[1,0,0,0],[0,0,0,0],[9E9,9E9,9E9,9E9,9E9,9E9]];
    PERS robtarget P03W21_Trans    := [[0,0,0],[1,0,0,0],[0,0,0,0],[9E9,9E9,9E9,9E9,9E9,9E9]];
    PERS bool P03W22_Used := FALSE;
    PERS num  P03W22_SubType := 0;
    PERS num  P03W22_ToolSel := 0;
    PERS num  P03W22_LenMM := 0;
    PERS robtarget P03W22_ArcStart := [[0,0,0],[1,0,0,0],[0,0,0,0],[9E9,9E9,9E9,9E9,9E9,9E9]];
    PERS robtarget P03W22_ArcEnd   := [[0,0,0],[1,0,0,0],[0,0,0,0],[9E9,9E9,9E9,9E9,9E9,9E9]];
    PERS robtarget P03W22_Approach := [[0,0,0],[1,0,0,0],[0,0,0,0],[9E9,9E9,9E9,9E9,9E9,9E9]];
    PERS robtarget P03W22_Retract  := [[0,0,0],[1,0,0,0],[0,0,0,0],[9E9,9E9,9E9,9E9,9E9,9E9]];
    PERS robtarget P03W22_Trans    := [[0,0,0],[1,0,0,0],[0,0,0,0],[9E9,9E9,9E9,9E9,9E9,9E9]];
    PERS bool P03W23_Used := FALSE;
    PERS num  P03W23_SubType := 0;
    PERS num  P03W23_ToolSel := 0;
    PERS num  P03W23_LenMM := 0;
    PERS robtarget P03W23_ArcStart := [[0,0,0],[1,0,0,0],[0,0,0,0],[9E9,9E9,9E9,9E9,9E9,9E9]];
    PERS robtarget P03W23_ArcEnd   := [[0,0,0],[1,0,0,0],[0,0,0,0],[9E9,9E9,9E9,9E9,9E9,9E9]];
    PERS robtarget P03W23_Approach := [[0,0,0],[1,0,0,0],[0,0,0,0],[9E9,9E9,9E9,9E9,9E9,9E9]];
    PERS robtarget P03W23_Retract  := [[0,0,0],[1,0,0,0],[0,0,0,0],[9E9,9E9,9E9,9E9,9E9,9E9]];
    PERS robtarget P03W23_Trans    := [[0,0,0],[1,0,0,0],[0,0,0,0],[9E9,9E9,9E9,9E9,9E9,9E9]];
    PERS bool P03W24_Used := FALSE;
    PERS num  P03W24_SubType := 0;
    PERS num  P03W24_ToolSel := 0;
    PERS num  P03W24_LenMM := 0;
    PERS robtarget P03W24_ArcStart := [[0,0,0],[1,0,0,0],[0,0,0,0],[9E9,9E9,9E9,9E9,9E9,9E9]];
    PERS robtarget P03W24_ArcEnd   := [[0,0,0],[1,0,0,0],[0,0,0,0],[9E9,9E9,9E9,9E9,9E9,9E9]];
    PERS robtarget P03W24_Approach := [[0,0,0],[1,0,0,0],[0,0,0,0],[9E9,9E9,9E9,9E9,9E9,9E9]];
    PERS robtarget P03W24_Retract  := [[0,0,0],[1,0,0,0],[0,0,0,0],[9E9,9E9,9E9,9E9,9E9,9E9]];
    PERS robtarget P03W24_Trans    := [[0,0,0],[1,0,0,0],[0,0,0,0],[9E9,9E9,9E9,9E9,9E9,9E9]];
    PERS bool P03W25_Used := FALSE;
    PERS num  P03W25_SubType := 0;
    PERS num  P03W25_ToolSel := 0;
    PERS num  P03W25_LenMM := 0;
    PERS robtarget P03W25_ArcStart := [[0,0,0],[1,0,0,0],[0,0,0,0],[9E9,9E9,9E9,9E9,9E9,9E9]];
    PERS robtarget P03W25_ArcEnd   := [[0,0,0],[1,0,0,0],[0,0,0,0],[9E9,9E9,9E9,9E9,9E9,9E9]];
    PERS robtarget P03W25_Approach := [[0,0,0],[1,0,0,0],[0,0,0,0],[9E9,9E9,9E9,9E9,9E9,9E9]];
    PERS robtarget P03W25_Retract  := [[0,0,0],[1,0,0,0],[0,0,0,0],[9E9,9E9,9E9,9E9,9E9,9E9]];
    PERS robtarget P03W25_Trans    := [[0,0,0],[1,0,0,0],[0,0,0,0],[9E9,9E9,9E9,9E9,9E9,9E9]];
    PERS bool P03W26_Used := FALSE;
    PERS num  P03W26_SubType := 0;
    PERS num  P03W26_ToolSel := 0;
    PERS num  P03W26_LenMM := 0;
    PERS robtarget P03W26_ArcStart := [[0,0,0],[1,0,0,0],[0,0,0,0],[9E9,9E9,9E9,9E9,9E9,9E9]];
    PERS robtarget P03W26_ArcEnd   := [[0,0,0],[1,0,0,0],[0,0,0,0],[9E9,9E9,9E9,9E9,9E9,9E9]];
    PERS robtarget P03W26_Approach := [[0,0,0],[1,0,0,0],[0,0,0,0],[9E9,9E9,9E9,9E9,9E9,9E9]];
    PERS robtarget P03W26_Retract  := [[0,0,0],[1,0,0,0],[0,0,0,0],[9E9,9E9,9E9,9E9,9E9,9E9]];
    PERS robtarget P03W26_Trans    := [[0,0,0],[1,0,0,0],[0,0,0,0],[9E9,9E9,9E9,9E9,9E9,9E9]];
    PERS bool P03W27_Used := FALSE;
    PERS num  P03W27_SubType := 0;
    PERS num  P03W27_ToolSel := 0;
    PERS num  P03W27_LenMM := 0;
    PERS robtarget P03W27_ArcStart := [[0,0,0],[1,0,0,0],[0,0,0,0],[9E9,9E9,9E9,9E9,9E9,9E9]];
    PERS robtarget P03W27_ArcEnd   := [[0,0,0],[1,0,0,0],[0,0,0,0],[9E9,9E9,9E9,9E9,9E9,9E9]];
    PERS robtarget P03W27_Approach := [[0,0,0],[1,0,0,0],[0,0,0,0],[9E9,9E9,9E9,9E9,9E9,9E9]];
    PERS robtarget P03W27_Retract  := [[0,0,0],[1,0,0,0],[0,0,0,0],[9E9,9E9,9E9,9E9,9E9,9E9]];
    PERS robtarget P03W27_Trans    := [[0,0,0],[1,0,0,0],[0,0,0,0],[9E9,9E9,9E9,9E9,9E9,9E9]];
    PERS bool P03W28_Used := FALSE;
    PERS num  P03W28_SubType := 0;
    PERS num  P03W28_ToolSel := 0;
    PERS num  P03W28_LenMM := 0;
    PERS robtarget P03W28_ArcStart := [[0,0,0],[1,0,0,0],[0,0,0,0],[9E9,9E9,9E9,9E9,9E9,9E9]];
    PERS robtarget P03W28_ArcEnd   := [[0,0,0],[1,0,0,0],[0,0,0,0],[9E9,9E9,9E9,9E9,9E9,9E9]];
    PERS robtarget P03W28_Approach := [[0,0,0],[1,0,0,0],[0,0,0,0],[9E9,9E9,9E9,9E9,9E9,9E9]];
    PERS robtarget P03W28_Retract  := [[0,0,0],[1,0,0,0],[0,0,0,0],[9E9,9E9,9E9,9E9,9E9,9E9]];
    PERS robtarget P03W28_Trans    := [[0,0,0],[1,0,0,0],[0,0,0,0],[9E9,9E9,9E9,9E9,9E9,9E9]];
    PERS bool P03W29_Used := FALSE;
    PERS num  P03W29_SubType := 0;
    PERS num  P03W29_ToolSel := 0;
    PERS num  P03W29_LenMM := 0;
    PERS robtarget P03W29_ArcStart := [[0,0,0],[1,0,0,0],[0,0,0,0],[9E9,9E9,9E9,9E9,9E9,9E9]];
    PERS robtarget P03W29_ArcEnd   := [[0,0,0],[1,0,0,0],[0,0,0,0],[9E9,9E9,9E9,9E9,9E9,9E9]];
    PERS robtarget P03W29_Approach := [[0,0,0],[1,0,0,0],[0,0,0,0],[9E9,9E9,9E9,9E9,9E9,9E9]];
    PERS robtarget P03W29_Retract  := [[0,0,0],[1,0,0,0],[0,0,0,0],[9E9,9E9,9E9,9E9,9E9,9E9]];
    PERS robtarget P03W29_Trans    := [[0,0,0],[1,0,0,0],[0,0,0,0],[9E9,9E9,9E9,9E9,9E9,9E9]];
    PERS bool P03W30_Used := FALSE;
    PERS num  P03W30_SubType := 0;
    PERS num  P03W30_ToolSel := 0;
    PERS num  P03W30_LenMM := 0;
    PERS robtarget P03W30_ArcStart := [[0,0,0],[1,0,0,0],[0,0,0,0],[9E9,9E9,9E9,9E9,9E9,9E9]];
    PERS robtarget P03W30_ArcEnd   := [[0,0,0],[1,0,0,0],[0,0,0,0],[9E9,9E9,9E9,9E9,9E9,9E9]];
    PERS robtarget P03W30_Approach := [[0,0,0],[1,0,0,0],[0,0,0,0],[9E9,9E9,9E9,9E9,9E9,9E9]];
    PERS robtarget P03W30_Retract  := [[0,0,0],[1,0,0,0],[0,0,0,0],[9E9,9E9,9E9,9E9,9E9,9E9]];
    PERS robtarget P03W30_Trans    := [[0,0,0],[1,0,0,0],[0,0,0,0],[9E9,9E9,9E9,9E9,9E9,9E9]];

    ! ---- P04 weld slots ----
    PERS bool P04W01_Used := FALSE;
    PERS num  P04W01_SubType := 0;
    PERS num  P04W01_ToolSel := 0;
    PERS num  P04W01_LenMM := 0;
    PERS robtarget P04W01_ArcStart := [[0,0,0],[1,0,0,0],[0,0,0,0],[9E9,9E9,9E9,9E9,9E9,9E9]];
    PERS robtarget P04W01_ArcEnd   := [[0,0,0],[1,0,0,0],[0,0,0,0],[9E9,9E9,9E9,9E9,9E9,9E9]];
    PERS robtarget P04W01_Approach := [[0,0,0],[1,0,0,0],[0,0,0,0],[9E9,9E9,9E9,9E9,9E9,9E9]];
    PERS robtarget P04W01_Retract  := [[0,0,0],[1,0,0,0],[0,0,0,0],[9E9,9E9,9E9,9E9,9E9,9E9]];
    PERS robtarget P04W01_Trans    := [[0,0,0],[1,0,0,0],[0,0,0,0],[9E9,9E9,9E9,9E9,9E9,9E9]];
    PERS bool P04W02_Used := FALSE;
    PERS num  P04W02_SubType := 0;
    PERS num  P04W02_ToolSel := 0;
    PERS num  P04W02_LenMM := 0;
    PERS robtarget P04W02_ArcStart := [[0,0,0],[1,0,0,0],[0,0,0,0],[9E9,9E9,9E9,9E9,9E9,9E9]];
    PERS robtarget P04W02_ArcEnd   := [[0,0,0],[1,0,0,0],[0,0,0,0],[9E9,9E9,9E9,9E9,9E9,9E9]];
    PERS robtarget P04W02_Approach := [[0,0,0],[1,0,0,0],[0,0,0,0],[9E9,9E9,9E9,9E9,9E9,9E9]];
    PERS robtarget P04W02_Retract  := [[0,0,0],[1,0,0,0],[0,0,0,0],[9E9,9E9,9E9,9E9,9E9,9E9]];
    PERS robtarget P04W02_Trans    := [[0,0,0],[1,0,0,0],[0,0,0,0],[9E9,9E9,9E9,9E9,9E9,9E9]];
    PERS bool P04W03_Used := FALSE;
    PERS num  P04W03_SubType := 0;
    PERS num  P04W03_ToolSel := 0;
    PERS num  P04W03_LenMM := 0;
    PERS robtarget P04W03_ArcStart := [[0,0,0],[1,0,0,0],[0,0,0,0],[9E9,9E9,9E9,9E9,9E9,9E9]];
    PERS robtarget P04W03_ArcEnd   := [[0,0,0],[1,0,0,0],[0,0,0,0],[9E9,9E9,9E9,9E9,9E9,9E9]];
    PERS robtarget P04W03_Approach := [[0,0,0],[1,0,0,0],[0,0,0,0],[9E9,9E9,9E9,9E9,9E9,9E9]];
    PERS robtarget P04W03_Retract  := [[0,0,0],[1,0,0,0],[0,0,0,0],[9E9,9E9,9E9,9E9,9E9,9E9]];
    PERS robtarget P04W03_Trans    := [[0,0,0],[1,0,0,0],[0,0,0,0],[9E9,9E9,9E9,9E9,9E9,9E9]];
    PERS bool P04W04_Used := FALSE;
    PERS num  P04W04_SubType := 0;
    PERS num  P04W04_ToolSel := 0;
    PERS num  P04W04_LenMM := 0;
    PERS robtarget P04W04_ArcStart := [[0,0,0],[1,0,0,0],[0,0,0,0],[9E9,9E9,9E9,9E9,9E9,9E9]];
    PERS robtarget P04W04_ArcEnd   := [[0,0,0],[1,0,0,0],[0,0,0,0],[9E9,9E9,9E9,9E9,9E9,9E9]];
    PERS robtarget P04W04_Approach := [[0,0,0],[1,0,0,0],[0,0,0,0],[9E9,9E9,9E9,9E9,9E9,9E9]];
    PERS robtarget P04W04_Retract  := [[0,0,0],[1,0,0,0],[0,0,0,0],[9E9,9E9,9E9,9E9,9E9,9E9]];
    PERS robtarget P04W04_Trans    := [[0,0,0],[1,0,0,0],[0,0,0,0],[9E9,9E9,9E9,9E9,9E9,9E9]];
    PERS bool P04W05_Used := FALSE;
    PERS num  P04W05_SubType := 0;
    PERS num  P04W05_ToolSel := 0;
    PERS num  P04W05_LenMM := 0;
    PERS robtarget P04W05_ArcStart := [[0,0,0],[1,0,0,0],[0,0,0,0],[9E9,9E9,9E9,9E9,9E9,9E9]];
    PERS robtarget P04W05_ArcEnd   := [[0,0,0],[1,0,0,0],[0,0,0,0],[9E9,9E9,9E9,9E9,9E9,9E9]];
    PERS robtarget P04W05_Approach := [[0,0,0],[1,0,0,0],[0,0,0,0],[9E9,9E9,9E9,9E9,9E9,9E9]];
    PERS robtarget P04W05_Retract  := [[0,0,0],[1,0,0,0],[0,0,0,0],[9E9,9E9,9E9,9E9,9E9,9E9]];
    PERS robtarget P04W05_Trans    := [[0,0,0],[1,0,0,0],[0,0,0,0],[9E9,9E9,9E9,9E9,9E9,9E9]];
    PERS bool P04W06_Used := FALSE;
    PERS num  P04W06_SubType := 0;
    PERS num  P04W06_ToolSel := 0;
    PERS num  P04W06_LenMM := 0;
    PERS robtarget P04W06_ArcStart := [[0,0,0],[1,0,0,0],[0,0,0,0],[9E9,9E9,9E9,9E9,9E9,9E9]];
    PERS robtarget P04W06_ArcEnd   := [[0,0,0],[1,0,0,0],[0,0,0,0],[9E9,9E9,9E9,9E9,9E9,9E9]];
    PERS robtarget P04W06_Approach := [[0,0,0],[1,0,0,0],[0,0,0,0],[9E9,9E9,9E9,9E9,9E9,9E9]];
    PERS robtarget P04W06_Retract  := [[0,0,0],[1,0,0,0],[0,0,0,0],[9E9,9E9,9E9,9E9,9E9,9E9]];
    PERS robtarget P04W06_Trans    := [[0,0,0],[1,0,0,0],[0,0,0,0],[9E9,9E9,9E9,9E9,9E9,9E9]];
    PERS bool P04W07_Used := FALSE;
    PERS num  P04W07_SubType := 0;
    PERS num  P04W07_ToolSel := 0;
    PERS num  P04W07_LenMM := 0;
    PERS robtarget P04W07_ArcStart := [[0,0,0],[1,0,0,0],[0,0,0,0],[9E9,9E9,9E9,9E9,9E9,9E9]];
    PERS robtarget P04W07_ArcEnd   := [[0,0,0],[1,0,0,0],[0,0,0,0],[9E9,9E9,9E9,9E9,9E9,9E9]];
    PERS robtarget P04W07_Approach := [[0,0,0],[1,0,0,0],[0,0,0,0],[9E9,9E9,9E9,9E9,9E9,9E9]];
    PERS robtarget P04W07_Retract  := [[0,0,0],[1,0,0,0],[0,0,0,0],[9E9,9E9,9E9,9E9,9E9,9E9]];
    PERS robtarget P04W07_Trans    := [[0,0,0],[1,0,0,0],[0,0,0,0],[9E9,9E9,9E9,9E9,9E9,9E9]];
    PERS bool P04W08_Used := FALSE;
    PERS num  P04W08_SubType := 0;
    PERS num  P04W08_ToolSel := 0;
    PERS num  P04W08_LenMM := 0;
    PERS robtarget P04W08_ArcStart := [[0,0,0],[1,0,0,0],[0,0,0,0],[9E9,9E9,9E9,9E9,9E9,9E9]];
    PERS robtarget P04W08_ArcEnd   := [[0,0,0],[1,0,0,0],[0,0,0,0],[9E9,9E9,9E9,9E9,9E9,9E9]];
    PERS robtarget P04W08_Approach := [[0,0,0],[1,0,0,0],[0,0,0,0],[9E9,9E9,9E9,9E9,9E9,9E9]];
    PERS robtarget P04W08_Retract  := [[0,0,0],[1,0,0,0],[0,0,0,0],[9E9,9E9,9E9,9E9,9E9,9E9]];
    PERS robtarget P04W08_Trans    := [[0,0,0],[1,0,0,0],[0,0,0,0],[9E9,9E9,9E9,9E9,9E9,9E9]];
    PERS bool P04W09_Used := FALSE;
    PERS num  P04W09_SubType := 0;
    PERS num  P04W09_ToolSel := 0;
    PERS num  P04W09_LenMM := 0;
    PERS robtarget P04W09_ArcStart := [[0,0,0],[1,0,0,0],[0,0,0,0],[9E9,9E9,9E9,9E9,9E9,9E9]];
    PERS robtarget P04W09_ArcEnd   := [[0,0,0],[1,0,0,0],[0,0,0,0],[9E9,9E9,9E9,9E9,9E9,9E9]];
    PERS robtarget P04W09_Approach := [[0,0,0],[1,0,0,0],[0,0,0,0],[9E9,9E9,9E9,9E9,9E9,9E9]];
    PERS robtarget P04W09_Retract  := [[0,0,0],[1,0,0,0],[0,0,0,0],[9E9,9E9,9E9,9E9,9E9,9E9]];
    PERS robtarget P04W09_Trans    := [[0,0,0],[1,0,0,0],[0,0,0,0],[9E9,9E9,9E9,9E9,9E9,9E9]];
    PERS bool P04W10_Used := FALSE;
    PERS num  P04W10_SubType := 0;
    PERS num  P04W10_ToolSel := 0;
    PERS num  P04W10_LenMM := 0;
    PERS robtarget P04W10_ArcStart := [[0,0,0],[1,0,0,0],[0,0,0,0],[9E9,9E9,9E9,9E9,9E9,9E9]];
    PERS robtarget P04W10_ArcEnd   := [[0,0,0],[1,0,0,0],[0,0,0,0],[9E9,9E9,9E9,9E9,9E9,9E9]];
    PERS robtarget P04W10_Approach := [[0,0,0],[1,0,0,0],[0,0,0,0],[9E9,9E9,9E9,9E9,9E9,9E9]];
    PERS robtarget P04W10_Retract  := [[0,0,0],[1,0,0,0],[0,0,0,0],[9E9,9E9,9E9,9E9,9E9,9E9]];
    PERS robtarget P04W10_Trans    := [[0,0,0],[1,0,0,0],[0,0,0,0],[9E9,9E9,9E9,9E9,9E9,9E9]];
    PERS bool P04W11_Used := FALSE;
    PERS num  P04W11_SubType := 0;
    PERS num  P04W11_ToolSel := 0;
    PERS num  P04W11_LenMM := 0;
    PERS robtarget P04W11_ArcStart := [[0,0,0],[1,0,0,0],[0,0,0,0],[9E9,9E9,9E9,9E9,9E9,9E9]];
    PERS robtarget P04W11_ArcEnd   := [[0,0,0],[1,0,0,0],[0,0,0,0],[9E9,9E9,9E9,9E9,9E9,9E9]];
    PERS robtarget P04W11_Approach := [[0,0,0],[1,0,0,0],[0,0,0,0],[9E9,9E9,9E9,9E9,9E9,9E9]];
    PERS robtarget P04W11_Retract  := [[0,0,0],[1,0,0,0],[0,0,0,0],[9E9,9E9,9E9,9E9,9E9,9E9]];
    PERS robtarget P04W11_Trans    := [[0,0,0],[1,0,0,0],[0,0,0,0],[9E9,9E9,9E9,9E9,9E9,9E9]];
    PERS bool P04W12_Used := FALSE;
    PERS num  P04W12_SubType := 0;
    PERS num  P04W12_ToolSel := 0;
    PERS num  P04W12_LenMM := 0;
    PERS robtarget P04W12_ArcStart := [[0,0,0],[1,0,0,0],[0,0,0,0],[9E9,9E9,9E9,9E9,9E9,9E9]];
    PERS robtarget P04W12_ArcEnd   := [[0,0,0],[1,0,0,0],[0,0,0,0],[9E9,9E9,9E9,9E9,9E9,9E9]];
    PERS robtarget P04W12_Approach := [[0,0,0],[1,0,0,0],[0,0,0,0],[9E9,9E9,9E9,9E9,9E9,9E9]];
    PERS robtarget P04W12_Retract  := [[0,0,0],[1,0,0,0],[0,0,0,0],[9E9,9E9,9E9,9E9,9E9,9E9]];
    PERS robtarget P04W12_Trans    := [[0,0,0],[1,0,0,0],[0,0,0,0],[9E9,9E9,9E9,9E9,9E9,9E9]];
    PERS bool P04W13_Used := FALSE;
    PERS num  P04W13_SubType := 0;
    PERS num  P04W13_ToolSel := 0;
    PERS num  P04W13_LenMM := 0;
    PERS robtarget P04W13_ArcStart := [[0,0,0],[1,0,0,0],[0,0,0,0],[9E9,9E9,9E9,9E9,9E9,9E9]];
    PERS robtarget P04W13_ArcEnd   := [[0,0,0],[1,0,0,0],[0,0,0,0],[9E9,9E9,9E9,9E9,9E9,9E9]];
    PERS robtarget P04W13_Approach := [[0,0,0],[1,0,0,0],[0,0,0,0],[9E9,9E9,9E9,9E9,9E9,9E9]];
    PERS robtarget P04W13_Retract  := [[0,0,0],[1,0,0,0],[0,0,0,0],[9E9,9E9,9E9,9E9,9E9,9E9]];
    PERS robtarget P04W13_Trans    := [[0,0,0],[1,0,0,0],[0,0,0,0],[9E9,9E9,9E9,9E9,9E9,9E9]];
    PERS bool P04W14_Used := FALSE;
    PERS num  P04W14_SubType := 0;
    PERS num  P04W14_ToolSel := 0;
    PERS num  P04W14_LenMM := 0;
    PERS robtarget P04W14_ArcStart := [[0,0,0],[1,0,0,0],[0,0,0,0],[9E9,9E9,9E9,9E9,9E9,9E9]];
    PERS robtarget P04W14_ArcEnd   := [[0,0,0],[1,0,0,0],[0,0,0,0],[9E9,9E9,9E9,9E9,9E9,9E9]];
    PERS robtarget P04W14_Approach := [[0,0,0],[1,0,0,0],[0,0,0,0],[9E9,9E9,9E9,9E9,9E9,9E9]];
    PERS robtarget P04W14_Retract  := [[0,0,0],[1,0,0,0],[0,0,0,0],[9E9,9E9,9E9,9E9,9E9,9E9]];
    PERS robtarget P04W14_Trans    := [[0,0,0],[1,0,0,0],[0,0,0,0],[9E9,9E9,9E9,9E9,9E9,9E9]];
    PERS bool P04W15_Used := FALSE;
    PERS num  P04W15_SubType := 0;
    PERS num  P04W15_ToolSel := 0;
    PERS num  P04W15_LenMM := 0;
    PERS robtarget P04W15_ArcStart := [[0,0,0],[1,0,0,0],[0,0,0,0],[9E9,9E9,9E9,9E9,9E9,9E9]];
    PERS robtarget P04W15_ArcEnd   := [[0,0,0],[1,0,0,0],[0,0,0,0],[9E9,9E9,9E9,9E9,9E9,9E9]];
    PERS robtarget P04W15_Approach := [[0,0,0],[1,0,0,0],[0,0,0,0],[9E9,9E9,9E9,9E9,9E9,9E9]];
    PERS robtarget P04W15_Retract  := [[0,0,0],[1,0,0,0],[0,0,0,0],[9E9,9E9,9E9,9E9,9E9,9E9]];
    PERS robtarget P04W15_Trans    := [[0,0,0],[1,0,0,0],[0,0,0,0],[9E9,9E9,9E9,9E9,9E9,9E9]];
    PERS bool P04W16_Used := FALSE;
    PERS num  P04W16_SubType := 0;
    PERS num  P04W16_ToolSel := 0;
    PERS num  P04W16_LenMM := 0;
    PERS robtarget P04W16_ArcStart := [[0,0,0],[1,0,0,0],[0,0,0,0],[9E9,9E9,9E9,9E9,9E9,9E9]];
    PERS robtarget P04W16_ArcEnd   := [[0,0,0],[1,0,0,0],[0,0,0,0],[9E9,9E9,9E9,9E9,9E9,9E9]];
    PERS robtarget P04W16_Approach := [[0,0,0],[1,0,0,0],[0,0,0,0],[9E9,9E9,9E9,9E9,9E9,9E9]];
    PERS robtarget P04W16_Retract  := [[0,0,0],[1,0,0,0],[0,0,0,0],[9E9,9E9,9E9,9E9,9E9,9E9]];
    PERS robtarget P04W16_Trans    := [[0,0,0],[1,0,0,0],[0,0,0,0],[9E9,9E9,9E9,9E9,9E9,9E9]];
    PERS bool P04W17_Used := FALSE;
    PERS num  P04W17_SubType := 0;
    PERS num  P04W17_ToolSel := 0;
    PERS num  P04W17_LenMM := 0;
    PERS robtarget P04W17_ArcStart := [[0,0,0],[1,0,0,0],[0,0,0,0],[9E9,9E9,9E9,9E9,9E9,9E9]];
    PERS robtarget P04W17_ArcEnd   := [[0,0,0],[1,0,0,0],[0,0,0,0],[9E9,9E9,9E9,9E9,9E9,9E9]];
    PERS robtarget P04W17_Approach := [[0,0,0],[1,0,0,0],[0,0,0,0],[9E9,9E9,9E9,9E9,9E9,9E9]];
    PERS robtarget P04W17_Retract  := [[0,0,0],[1,0,0,0],[0,0,0,0],[9E9,9E9,9E9,9E9,9E9,9E9]];
    PERS robtarget P04W17_Trans    := [[0,0,0],[1,0,0,0],[0,0,0,0],[9E9,9E9,9E9,9E9,9E9,9E9]];
    PERS bool P04W18_Used := FALSE;
    PERS num  P04W18_SubType := 0;
    PERS num  P04W18_ToolSel := 0;
    PERS num  P04W18_LenMM := 0;
    PERS robtarget P04W18_ArcStart := [[0,0,0],[1,0,0,0],[0,0,0,0],[9E9,9E9,9E9,9E9,9E9,9E9]];
    PERS robtarget P04W18_ArcEnd   := [[0,0,0],[1,0,0,0],[0,0,0,0],[9E9,9E9,9E9,9E9,9E9,9E9]];
    PERS robtarget P04W18_Approach := [[0,0,0],[1,0,0,0],[0,0,0,0],[9E9,9E9,9E9,9E9,9E9,9E9]];
    PERS robtarget P04W18_Retract  := [[0,0,0],[1,0,0,0],[0,0,0,0],[9E9,9E9,9E9,9E9,9E9,9E9]];
    PERS robtarget P04W18_Trans    := [[0,0,0],[1,0,0,0],[0,0,0,0],[9E9,9E9,9E9,9E9,9E9,9E9]];
    PERS bool P04W19_Used := FALSE;
    PERS num  P04W19_SubType := 0;
    PERS num  P04W19_ToolSel := 0;
    PERS num  P04W19_LenMM := 0;
    PERS robtarget P04W19_ArcStart := [[0,0,0],[1,0,0,0],[0,0,0,0],[9E9,9E9,9E9,9E9,9E9,9E9]];
    PERS robtarget P04W19_ArcEnd   := [[0,0,0],[1,0,0,0],[0,0,0,0],[9E9,9E9,9E9,9E9,9E9,9E9]];
    PERS robtarget P04W19_Approach := [[0,0,0],[1,0,0,0],[0,0,0,0],[9E9,9E9,9E9,9E9,9E9,9E9]];
    PERS robtarget P04W19_Retract  := [[0,0,0],[1,0,0,0],[0,0,0,0],[9E9,9E9,9E9,9E9,9E9,9E9]];
    PERS robtarget P04W19_Trans    := [[0,0,0],[1,0,0,0],[0,0,0,0],[9E9,9E9,9E9,9E9,9E9,9E9]];
    PERS bool P04W20_Used := FALSE;
    PERS num  P04W20_SubType := 0;
    PERS num  P04W20_ToolSel := 0;
    PERS num  P04W20_LenMM := 0;
    PERS robtarget P04W20_ArcStart := [[0,0,0],[1,0,0,0],[0,0,0,0],[9E9,9E9,9E9,9E9,9E9,9E9]];
    PERS robtarget P04W20_ArcEnd   := [[0,0,0],[1,0,0,0],[0,0,0,0],[9E9,9E9,9E9,9E9,9E9,9E9]];
    PERS robtarget P04W20_Approach := [[0,0,0],[1,0,0,0],[0,0,0,0],[9E9,9E9,9E9,9E9,9E9,9E9]];
    PERS robtarget P04W20_Retract  := [[0,0,0],[1,0,0,0],[0,0,0,0],[9E9,9E9,9E9,9E9,9E9,9E9]];
    PERS robtarget P04W20_Trans    := [[0,0,0],[1,0,0,0],[0,0,0,0],[9E9,9E9,9E9,9E9,9E9,9E9]];
    PERS bool P04W21_Used := FALSE;
    PERS num  P04W21_SubType := 0;
    PERS num  P04W21_ToolSel := 0;
    PERS num  P04W21_LenMM := 0;
    PERS robtarget P04W21_ArcStart := [[0,0,0],[1,0,0,0],[0,0,0,0],[9E9,9E9,9E9,9E9,9E9,9E9]];
    PERS robtarget P04W21_ArcEnd   := [[0,0,0],[1,0,0,0],[0,0,0,0],[9E9,9E9,9E9,9E9,9E9,9E9]];
    PERS robtarget P04W21_Approach := [[0,0,0],[1,0,0,0],[0,0,0,0],[9E9,9E9,9E9,9E9,9E9,9E9]];
    PERS robtarget P04W21_Retract  := [[0,0,0],[1,0,0,0],[0,0,0,0],[9E9,9E9,9E9,9E9,9E9,9E9]];
    PERS robtarget P04W21_Trans    := [[0,0,0],[1,0,0,0],[0,0,0,0],[9E9,9E9,9E9,9E9,9E9,9E9]];
    PERS bool P04W22_Used := FALSE;
    PERS num  P04W22_SubType := 0;
    PERS num  P04W22_ToolSel := 0;
    PERS num  P04W22_LenMM := 0;
    PERS robtarget P04W22_ArcStart := [[0,0,0],[1,0,0,0],[0,0,0,0],[9E9,9E9,9E9,9E9,9E9,9E9]];
    PERS robtarget P04W22_ArcEnd   := [[0,0,0],[1,0,0,0],[0,0,0,0],[9E9,9E9,9E9,9E9,9E9,9E9]];
    PERS robtarget P04W22_Approach := [[0,0,0],[1,0,0,0],[0,0,0,0],[9E9,9E9,9E9,9E9,9E9,9E9]];
    PERS robtarget P04W22_Retract  := [[0,0,0],[1,0,0,0],[0,0,0,0],[9E9,9E9,9E9,9E9,9E9,9E9]];
    PERS robtarget P04W22_Trans    := [[0,0,0],[1,0,0,0],[0,0,0,0],[9E9,9E9,9E9,9E9,9E9,9E9]];
    PERS bool P04W23_Used := FALSE;
    PERS num  P04W23_SubType := 0;
    PERS num  P04W23_ToolSel := 0;
    PERS num  P04W23_LenMM := 0;
    PERS robtarget P04W23_ArcStart := [[0,0,0],[1,0,0,0],[0,0,0,0],[9E9,9E9,9E9,9E9,9E9,9E9]];
    PERS robtarget P04W23_ArcEnd   := [[0,0,0],[1,0,0,0],[0,0,0,0],[9E9,9E9,9E9,9E9,9E9,9E9]];
    PERS robtarget P04W23_Approach := [[0,0,0],[1,0,0,0],[0,0,0,0],[9E9,9E9,9E9,9E9,9E9,9E9]];
    PERS robtarget P04W23_Retract  := [[0,0,0],[1,0,0,0],[0,0,0,0],[9E9,9E9,9E9,9E9,9E9,9E9]];
    PERS robtarget P04W23_Trans    := [[0,0,0],[1,0,0,0],[0,0,0,0],[9E9,9E9,9E9,9E9,9E9,9E9]];
    PERS bool P04W24_Used := FALSE;
    PERS num  P04W24_SubType := 0;
    PERS num  P04W24_ToolSel := 0;
    PERS num  P04W24_LenMM := 0;
    PERS robtarget P04W24_ArcStart := [[0,0,0],[1,0,0,0],[0,0,0,0],[9E9,9E9,9E9,9E9,9E9,9E9]];
    PERS robtarget P04W24_ArcEnd   := [[0,0,0],[1,0,0,0],[0,0,0,0],[9E9,9E9,9E9,9E9,9E9,9E9]];
    PERS robtarget P04W24_Approach := [[0,0,0],[1,0,0,0],[0,0,0,0],[9E9,9E9,9E9,9E9,9E9,9E9]];
    PERS robtarget P04W24_Retract  := [[0,0,0],[1,0,0,0],[0,0,0,0],[9E9,9E9,9E9,9E9,9E9,9E9]];
    PERS robtarget P04W24_Trans    := [[0,0,0],[1,0,0,0],[0,0,0,0],[9E9,9E9,9E9,9E9,9E9,9E9]];
    PERS bool P04W25_Used := FALSE;
    PERS num  P04W25_SubType := 0;
    PERS num  P04W25_ToolSel := 0;
    PERS num  P04W25_LenMM := 0;
    PERS robtarget P04W25_ArcStart := [[0,0,0],[1,0,0,0],[0,0,0,0],[9E9,9E9,9E9,9E9,9E9,9E9]];
    PERS robtarget P04W25_ArcEnd   := [[0,0,0],[1,0,0,0],[0,0,0,0],[9E9,9E9,9E9,9E9,9E9,9E9]];
    PERS robtarget P04W25_Approach := [[0,0,0],[1,0,0,0],[0,0,0,0],[9E9,9E9,9E9,9E9,9E9,9E9]];
    PERS robtarget P04W25_Retract  := [[0,0,0],[1,0,0,0],[0,0,0,0],[9E9,9E9,9E9,9E9,9E9,9E9]];
    PERS robtarget P04W25_Trans    := [[0,0,0],[1,0,0,0],[0,0,0,0],[9E9,9E9,9E9,9E9,9E9,9E9]];
    PERS bool P04W26_Used := FALSE;
    PERS num  P04W26_SubType := 0;
    PERS num  P04W26_ToolSel := 0;
    PERS num  P04W26_LenMM := 0;
    PERS robtarget P04W26_ArcStart := [[0,0,0],[1,0,0,0],[0,0,0,0],[9E9,9E9,9E9,9E9,9E9,9E9]];
    PERS robtarget P04W26_ArcEnd   := [[0,0,0],[1,0,0,0],[0,0,0,0],[9E9,9E9,9E9,9E9,9E9,9E9]];
    PERS robtarget P04W26_Approach := [[0,0,0],[1,0,0,0],[0,0,0,0],[9E9,9E9,9E9,9E9,9E9,9E9]];
    PERS robtarget P04W26_Retract  := [[0,0,0],[1,0,0,0],[0,0,0,0],[9E9,9E9,9E9,9E9,9E9,9E9]];
    PERS robtarget P04W26_Trans    := [[0,0,0],[1,0,0,0],[0,0,0,0],[9E9,9E9,9E9,9E9,9E9,9E9]];
    PERS bool P04W27_Used := FALSE;
    PERS num  P04W27_SubType := 0;
    PERS num  P04W27_ToolSel := 0;
    PERS num  P04W27_LenMM := 0;
    PERS robtarget P04W27_ArcStart := [[0,0,0],[1,0,0,0],[0,0,0,0],[9E9,9E9,9E9,9E9,9E9,9E9]];
    PERS robtarget P04W27_ArcEnd   := [[0,0,0],[1,0,0,0],[0,0,0,0],[9E9,9E9,9E9,9E9,9E9,9E9]];
    PERS robtarget P04W27_Approach := [[0,0,0],[1,0,0,0],[0,0,0,0],[9E9,9E9,9E9,9E9,9E9,9E9]];
    PERS robtarget P04W27_Retract  := [[0,0,0],[1,0,0,0],[0,0,0,0],[9E9,9E9,9E9,9E9,9E9,9E9]];
    PERS robtarget P04W27_Trans    := [[0,0,0],[1,0,0,0],[0,0,0,0],[9E9,9E9,9E9,9E9,9E9,9E9]];
    PERS bool P04W28_Used := FALSE;
    PERS num  P04W28_SubType := 0;
    PERS num  P04W28_ToolSel := 0;
    PERS num  P04W28_LenMM := 0;
    PERS robtarget P04W28_ArcStart := [[0,0,0],[1,0,0,0],[0,0,0,0],[9E9,9E9,9E9,9E9,9E9,9E9]];
    PERS robtarget P04W28_ArcEnd   := [[0,0,0],[1,0,0,0],[0,0,0,0],[9E9,9E9,9E9,9E9,9E9,9E9]];
    PERS robtarget P04W28_Approach := [[0,0,0],[1,0,0,0],[0,0,0,0],[9E9,9E9,9E9,9E9,9E9,9E9]];
    PERS robtarget P04W28_Retract  := [[0,0,0],[1,0,0,0],[0,0,0,0],[9E9,9E9,9E9,9E9,9E9,9E9]];
    PERS robtarget P04W28_Trans    := [[0,0,0],[1,0,0,0],[0,0,0,0],[9E9,9E9,9E9,9E9,9E9,9E9]];
    PERS bool P04W29_Used := FALSE;
    PERS num  P04W29_SubType := 0;
    PERS num  P04W29_ToolSel := 0;
    PERS num  P04W29_LenMM := 0;
    PERS robtarget P04W29_ArcStart := [[0,0,0],[1,0,0,0],[0,0,0,0],[9E9,9E9,9E9,9E9,9E9,9E9]];
    PERS robtarget P04W29_ArcEnd   := [[0,0,0],[1,0,0,0],[0,0,0,0],[9E9,9E9,9E9,9E9,9E9,9E9]];
    PERS robtarget P04W29_Approach := [[0,0,0],[1,0,0,0],[0,0,0,0],[9E9,9E9,9E9,9E9,9E9,9E9]];
    PERS robtarget P04W29_Retract  := [[0,0,0],[1,0,0,0],[0,0,0,0],[9E9,9E9,9E9,9E9,9E9,9E9]];
    PERS robtarget P04W29_Trans    := [[0,0,0],[1,0,0,0],[0,0,0,0],[9E9,9E9,9E9,9E9,9E9,9E9]];
    PERS bool P04W30_Used := FALSE;
    PERS num  P04W30_SubType := 0;
    PERS num  P04W30_ToolSel := 0;
    PERS num  P04W30_LenMM := 0;
    PERS robtarget P04W30_ArcStart := [[0,0,0],[1,0,0,0],[0,0,0,0],[9E9,9E9,9E9,9E9,9E9,9E9]];
    PERS robtarget P04W30_ArcEnd   := [[0,0,0],[1,0,0,0],[0,0,0,0],[9E9,9E9,9E9,9E9,9E9,9E9]];
    PERS robtarget P04W30_Approach := [[0,0,0],[1,0,0,0],[0,0,0,0],[9E9,9E9,9E9,9E9,9E9,9E9]];
    PERS robtarget P04W30_Retract  := [[0,0,0],[1,0,0,0],[0,0,0,0],[9E9,9E9,9E9,9E9,9E9,9E9]];
    PERS robtarget P04W30_Trans    := [[0,0,0],[1,0,0,0],[0,0,0,0],[9E9,9E9,9E9,9E9,9E9,9E9]];

